LIN {X 0,Y 446.479,Z 402.372,A -85,B 0,C 180,E1 -8668.18,E2 -8668.18} C_VEL
LIN {X 0,Y 446.415,Z 402.374,A -85,B 0,C 180,E1 -8671.301,E2 -8671.301} C_VEL
LIN {X 0,Y 446.426,Z 402.376,A -85,B 0,C 180,E1 -8674.524,E2 -8674.524} C_VEL
LIN {X 0,Y 446.431,Z 402.379,A -85,B 0,C 180,E1 -8678.083,E2 -8678.083} C_VEL
LIN {X 0,Y 446.448,Z 402.406,A -85,B 0,C 180,E1 -8680.922,E2 -8680.922} C_VEL
LIN {X 0,Y 446.858,Z 405.436,A -85,B 0,C 180,E1 -8683.79,E2 -8683.79} C_VEL
LIN {X 0,Y 447.262,Z 408.259,A -85,B 0,C 180,E1 -8686.288,E2 -8686.288} C_VEL
LIN {X 0,Y 447.316,Z 411.248,A -85,B 0,C 180,E1 -8688.71,E2 -8688.71} C_VEL
LIN {X 0,Y 447.118,Z 415.361,A -85,B 0,C 180,E1 -8691.807,E2 -8691.807} C_VEL
LIN {X 0,Y 446.835,Z 419.717,A -85,B 0,C 180,E1 -8694.874,E2 -8694.874} C_VEL
LIN {X 0,Y 446.566,Z 423.896,A -85,B 0,C 180,E1 -8697.651,E2 -8697.651} C_VEL
LIN {X 0,Y 446.285,Z 428.788,A -85,B 0,C 180,E1 -8700.78,E2 -8700.78} C_VEL
LIN {X 0,Y 446.043,Z 433.937,A -85,B 0,C 180,E1 -8703.912,E2 -8703.912} C_VEL
LIN {X 0,Y 445.834,Z 438.832,A -85,B 0,C 180,E1 -8706.791,E2 -8706.791} C_VEL
LIN {X 0,Y 445.676,Z 443.934,A -85,B 0,C 180,E1 -8709.701,E2 -8709.701} C_VEL
LIN {X 0,Y 445.528,Z 449.059,A -85,B 0,C 180,E1 -8712.56,E2 -8712.56} C_VEL
LIN {X 0,Y 445.534,Z 451.508,A -85,B 0,C 180,E1 -8713.873,E2 -8713.873} C_VEL
LIN {X 0,Y 447.627,Z 463.278,A -85,B 0,C 180,E1 -8714.29,E2 -8714.29} C_VEL
LIN {X 0,Y 449.274,Z 475.733,A -85,B 0,C 180,E1 -8714.868,E2 -8714.868} C_VEL
LIN {X 0,Y 448.649,Z 488.448,A -85,B 0,C 180,E1 -8715.601,E2 -8715.601} C_VEL
LIN {X 0,Y 448.166,Z 497.727,A -85,B 0,C 180,E1 -8716.28,E2 -8716.28} C_VEL
LIN {X 0,Y 447.678,Z 506.19,A -85,B 0,C 180,E1 -8717.024,E2 -8717.024} C_VEL
LIN {X 0,Y 447.323,Z 513.287,A -85,B 0,C 180,E1 -8717.755,E2 -8717.755} C_VEL
LIN {X 0,Y 446.729,Z 522.426,A -85,B 0,C 180,E1 -8718.889,E2 -8718.889} C_VEL
LIN {X 0,Y 446.396,Z 528.63,A -85,B 0,C 180,E1 -8719.798,E2 -8719.798} C_VEL
LIN {X 0,Y 446.041,Z 535.168,A -85,B 0,C 180,E1 -8720.935,E2 -8720.935} C_VEL
LIN {X 0,Y 445.849,Z 539.67,A -85,B 0,C 180,E1 -8721.844,E2 -8721.844} C_VEL
LIN {X 0,Y 445.584,Z 545.162,A -85,B 0,C 180,E1 -8723.207,E2 -8723.207} C_VEL
LIN {X 0,Y 445.49,Z 549.484,A -85,B 0,C 180,E1 -8724.569,E2 -8724.569} C_VEL
LIN {X 0,Y 445.419,Z 551.848,A -85,B 0,C 180,E1 -8725.475,E2 -8725.475} C_VEL
LIN {X 0,Y 445.434,Z 555.032,A -85,B 0,C 180,E1 -8727.287,E2 -8727.287} C_VEL
LIN {X 0,Y 445.356,Z 556.087,A -85,B 0,C 180,E1 -8728.191,E2 -8728.191} C_VEL
LIN {X 0,Y 445.339,Z 556.674,A -85,B 0,C 180,E1 -8729.096,E2 -8729.096} C_VEL
LIN {X 0,Y 445.339,Z 556.674,A -85,B 0,C 180,E1 -8730.904,E2 -8730.904} C_VEL
LIN {X 0,Y 445.356,Z 556.087,A -85,B 0,C 180,E1 -8731.809,E2 -8731.809} C_VEL
LIN {X 0,Y 445.434,Z 555.032,A -85,B 0,C 180,E1 -8732.713,E2 -8732.713} C_VEL
LIN {X 0,Y 445.419,Z 551.848,A -85,B 0,C 180,E1 -8734.525,E2 -8734.525} C_VEL
LIN {X 0,Y 445.491,Z 547.64,A -85,B 0,C 180,E1 -8736.069,E2 -8736.069} C_VEL
LIN {X 0,Y 445.668,Z 543.501,A -85,B 0,C 180,E1 -8737.247,E2 -8737.247} C_VEL
LIN {X 0,Y 445.963,Z 537.48,A -85,B 0,C 180,E1 -8738.61,E2 -8738.61} C_VEL
LIN {X 0,Y 446.227,Z 531.382,A -85,B 0,C 180,E1 -8739.748,E2 -8739.748} C_VEL
LIN {X 0,Y 446.532,Z 525.681,A -85,B 0,C 180,E1 -8740.657,E2 -8740.657} C_VEL
LIN {X 0,Y 447.064,Z 517.126,A -85,B 0,C 180,E1 -8741.792,E2 -8741.792} C_VEL
LIN {X 0,Y 447.555,Z 508.945,A -85,B 0,C 180,E1 -8742.7,E2 -8742.7} C_VEL
LIN {X 0,Y 447.937,Z 500.62,A -85,B 0,C 180,E1 -8743.48,E2 -8743.48} C_VEL
LIN {X 0,Y 448.472,Z 491.713,A -85,B 0,C 180,E1 -8744.173,E2 -8744.173} C_VEL
LIN {X 0,Y 448.975,Z 481.953,A -85,B 0,C 180,E1 -8744.794,E2 -8744.794} C_VEL
LIN {X 0,Y 449.187,Z 474.443,A -85,B 0,C 180,E1 -8745.193,E2 -8745.193} C_VEL
LIN {X 0,Y 447.597,Z 463.013,A -85,B 0,C 180,E1 -8745.72,E2 -8745.72} C_VEL
LIN {X 0,Y 445.662,Z 452.543,A -85,B 0,C 180,E1 -8746.094,E2 -8746.094} C_VEL
LIN {X 0,Y 445.535,Z 451.449,A -85,B 0,C 180,E1 -8746.157,E2 -8746.157} C_VEL
LIN {X 0,Y 445.643,Z 445.63,A -85,B 0,C 180,E1 -8749.34,E2 -8749.34} C_VEL
LIN {X 0,Y 445.775,Z 440.518,A -85,B 0,C 180,E1 -8752.233,E2 -8752.233} C_VEL
LIN {X 0,Y 445.947,Z 435.451,A -85,B 0,C 180,E1 -8755.183,E2 -8755.183} C_VEL
LIN {X 0,Y 446.216,Z 430.442,A -85,B 0,C 180,E1 -8758.196,E2 -8758.196} C_VEL
LIN {X 0,Y 446.487,Z 425.503,A -85,B 0,C 180,E1 -8761.294,E2 -8761.294} C_VEL
LIN {X 0,Y 446.768,Z 420.645,A -85,B 0,C 180,E1 -8764.492,E2 -8764.492} C_VEL
LIN {X 0,Y 447.005,Z 417.453,A -85,B 0,C 180,E1 -8766.693,E2 -8766.693} C_VEL
LIN {X 0,Y 447.227,Z 413.373,A -85,B 0,C 180,E1 -8769.644,E2 -8769.644} C_VEL
LIN {X 0,Y 447.365,Z 409.716,A -85,B 0,C 180,E1 -8772.493,E2 -8772.493} C_VEL
LIN {X 0,Y 447.061,Z 406.738,A -85,B 0,C 180,E1 -8775.024,E2 -8775.024} C_VEL
LIN {X 0,Y 446.515,Z 402.871,A -85,B 0,C 180,E1 -8778.618,E2 -8778.618} C_VEL
LIN {X 0,Y 446.448,Z 402.407,A -85,B 0,C 180,E1 -8779.078,E2 -8779.078} C_VEL
LIN {X 0,Y 446.431,Z 402.378,A -85,B 0,C 180,E1 -8781.917,E2 -8781.917} C_VEL
LIN {X 0,Y 446.426,Z 402.378,A -85,B 0,C 180,E1 -8785.476,E2 -8785.476} C_VEL
LIN {X 0,Y 446.415,Z 402.374,A -85,B 0,C 180,E1 -8788.699,E2 -8788.699} C_VEL
LIN {X 0,Y 446.479,Z 402.372,A -85,B 0,C 180,E1 -8791.82,E2 -8791.82} C_VEL
LIN {X 0,Y 446.451,Z 402.369,A -85,B 0,C 180,E1 -8794.847,E2 -8794.847} C_VEL
LIN {X 0,Y 446.441,Z 402.373,A -85,B 0,C 180,E1 -8798.244,E2 -8798.244} C_VEL
LIN {X 0,Y 446.451,Z 402.375,A -85,B 0,C 180,E1 -8801.648,E2 -8801.648} C_VEL
LIN {X 0,Y 446.509,Z 402.362,A -85,B 0,C 180,E1 -8804.479,E2 -8804.479} C_VEL
LIN {X 0,Y 446.51,Z 402.363,A -85,B 0,C 180,E1 -8808.192,E2 -8808.192} C_VEL
LIN {X 0,Y 446.592,Z 402.356,A -85,B 0,C 180,E1 -8811.857,E2 -8811.857} C_VEL
LIN {X 0,Y 446.638,Z 402.345,A -85,B 0,C 180,E1 -8814.582,E2 -8814.582} C_VEL
LIN {X 0,Y 446.701,Z 402.343,A -85,B 0,C 180,E1 -8817.294,E2 -8817.294} C_VEL
LIN {X 0,Y 446.784,Z 402.329,A -85,B 0,C 180,E1 -8819.999,E2 -8819.999} C_VEL
LIN {X 0,Y 446.701,Z 402.338,A -85,B 0,C 180,E1 -8822.705,E2 -8822.705} C_VEL
LIN {X 0,Y 446.639,Z 402.345,A -85,B 0,C 180,E1 -8826.323,E2 -8826.323} C_VEL
LIN {X 0,Y 446.529,Z 402.363,A -85,B 0,C 180,E1 -8829.055,E2 -8829.055} C_VEL
LIN {X 0,Y 446.514,Z 402.363,A -85,B 0,C 180,E1 -8832.729,E2 -8832.729} C_VEL
LIN {X 0,Y 446.487,Z 402.364,A -85,B 0,C 180,E1 -8836.228,E2 -8836.228} C_VEL
LIN {X 0,Y 446.46,Z 402.373,A -85,B 0,C 180,E1 -8839.303,E2 -8839.303} C_VEL
LIN {X 0,Y 446.408,Z 402.374,A -85,B 0,C 180,E1 -8842.2,E2 -8842.2} C_VEL
LIN {X 0,Y 446.449,Z 402.376,A -85,B 0,C 180,E1 -8845.152,E2 -8845.152} C_VEL
LIN {X 0,Y 446.475,Z 402.366,A -85,B 0,C 180,E1 -8848.179,E2 -8848.179} C_VEL
LIN {X 0,Y 446.411,Z 402.377,A -85,B 0,C 180,E1 -8851.3,E2 -8851.3} C_VEL
LIN {X 0,Y 446.422,Z 402.375,A -85,B 0,C 180,E1 -8854.523,E2 -8854.523} C_VEL
LIN {X 0,Y 446.43,Z 402.372,A -85,B 0,C 180,E1 -8858.083,E2 -8858.083} C_VEL
LIN {X 0,Y 446.439,Z 402.376,A -85,B 0,C 180,E1 -8860.921,E2 -8860.921} C_VEL
LIN {X 0,Y 446.437,Z 402.37,A -85,B 0,C 180,E1 -8863.841,E2 -8863.841} C_VEL
LIN {X 0,Y 446.413,Z 402.377,A -85,B 0,C 180,E1 -8866.401,E2 -8866.401} C_VEL
LIN {X 0,Y 446.444,Z 402.37,A -85,B 0,C 180,E1 -8869.803,E2 -8869.803} C_VEL
LIN {X 0,Y 446.421,Z 402.375,A -85,B 0,C 180,E1 -8872.123,E2 -8872.123} C_VEL
LIN {X 0,Y 446.424,Z 402.372,A -85,B 0,C 180,E1 -8875.477,E2 -8875.477} C_VEL
LIN {X 0,Y 446.411,Z 402.379,A -85,B 0,C 180,E1 -8878.7,E2 -8878.7} C_VEL
LIN {X 0,Y 446.479,Z 402.366,A -85,B 0,C 180,E1 -8881.822,E2 -8881.822} C_VEL
LIN {X 0,Y 446.453,Z 402.371,A -85,B 0,C 180,E1 -8884.848,E2 -8884.848} C_VEL
LIN {X 0,Y 446.443,Z 402.376,A -85,B 0,C 180,E1 -8888.245,E2 -8888.245} C_VEL
LIN {X 0,Y 446.453,Z 402.373,A -85,B 0,C 180,E1 -8891.649,E2 -8891.649} C_VEL
LIN {X 0,Y 446.503,Z 402.369,A -85,B 0,C 180,E1 -8894.48,E2 -8894.48} C_VEL
LIN {X 0,Y 446.514,Z 402.368,A -85,B 0,C 180,E1 -8898.193,E2 -8898.193} C_VEL
LIN {X 0,Y 446.596,Z 402.357,A -85,B 0,C 180,E1 -8901.858,E2 -8901.858} C_VEL
LIN {X 0,Y 446.643,Z 402.351,A -85,B 0,C 180,E1 -8904.583,E2 -8904.583} C_VEL
LIN {X 0,Y 446.622,Z 402.351,A -85,B 0,C 180,E1 -8907.011,E2 -8907.011} C_VEL
LIN {X 0,Y 446.104,Z 402.419,A -85,B 0,C 180,E1 -8907.764,E2 -8907.764} C_VEL
LIN {X 0,Y 443.288,Z 402.77,A -85,B 0,C 180,E1 -8908.987,E2 -8908.987} C_VEL
LIN {X 0,Y 440.801,Z 403.08,A -85,B 0,C 180,E1 -8909.974,E2 -8909.974} C_VEL
LIN {X 0,Y 439.712,Z 403.214,A -85,B 0,C 180,E1 -8910.737,E2 -8910.737} C_VEL
LIN {X 0,Y 439.618,Z 403.224,A -85,B 0,C 180,E1 -8910.996,E2 -8910.996} C_VEL
LIN {X 0,Y 439.653,Z 403.22,A -85,B 0,C 180,E1 -8912.749,E2 -8912.749} C_VEL
LIN {X 0,Y 439.615,Z 403.225,A -85,B 0,C 180,E1 -8916.425,E2 -8916.425} C_VEL
LIN {X 0,Y 439.496,Z 403.24,A -85,B 0,C 180,E1 -8919.201,E2 -8919.201} C_VEL
LIN {X 0,Y 439.461,Z 403.243,A -85,B 0,C 180,E1 -8922.937,E2 -8922.937} C_VEL
LIN {X 0,Y 439.443,Z 403.246,A -85,B 0,C 180,E1 -8926.349,E2 -8926.349} C_VEL
LIN {X 0,Y 439.398,Z 403.255,A -85,B 0,C 180,E1 -8929.626,E2 -8929.626} C_VEL
LIN {X 0,Y 439.36,Z 403.252,A -85,B 0,C 180,E1 -8932.575,E2 -8932.575} C_VEL
LIN {X 0,Y 439.401,Z 403.255,A -85,B 0,C 180,E1 -8935.584,E2 -8935.584} C_VEL
LIN {X 0,Y 439.412,Z 403.246,A -85,B 0,C 180,E1 -8938.673,E2 -8938.673} C_VEL
LIN {X 0,Y 439.365,Z 403.253,A -85,B 0,C 180,E1 -8942.03,E2 -8942.03} C_VEL
LIN {X 0,Y 439.39,Z 403.255,A -85,B 0,C 180,E1 -8945.34,E2 -8945.34} C_VEL
LIN {X 0,Y 439.383,Z 403.25,A -85,B 0,C 180,E1 -8948.594,E2 -8948.594} C_VEL
LIN {X 0,Y 439.382,Z 403.256,A -85,B 0,C 180,E1 -8951.257,E2 -8951.257} C_VEL
LIN {X 0,Y 439.398,Z 403.249,A -85,B 0,C 180,E1 -8954.728,E2 -8954.728} C_VEL
LIN {X 0,Y 439.39,Z 403.25,A -85,B 0,C 180,E1 -8957.796,E2 -8957.796} C_VEL
LIN {X 0,Y 439.417,Z 403.245,A -85,B 0,C 180,E1 -8960.227,E2 -8960.227} C_VEL
LIN {X 0,Y 439.368,Z 403.252,A -85,B 0,C 180,E1 -8963.713,E2 -8963.713} C_VEL
LIN {X 0,Y 439.365,Z 403.259,A -85,B 0,C 180,E1 -8967.054,E2 -8967.054} C_VEL
LIN {X 0,Y 439.387,Z 403.249,A -85,B 0,C 180,E1 -8970.275,E2 -8970.275} C_VEL
LIN {X 0,Y 439.424,Z 403.245,A -85,B 0,C 180,E1 -8973.589,E2 -8973.589} C_VEL
LIN {X 0,Y 439.377,Z 403.252,A -85,B 0,C 180,E1 -8976.43,E2 -8976.43} C_VEL
LIN {X 0,Y 439.379,Z 403.251,A -85,B 0,C 180,E1 -8979.397,E2 -8979.397} C_VEL
LIN {X 0,Y 439.422,Z 403.246,A -85,B 0,C 180,E1 -8982.31,E2 -8982.31} C_VEL
LIN {X 0,Y 439.44,Z 403.245,A -85,B 0,C 180,E1 -8985.174,E2 -8985.174} C_VEL
LIN {X 0,Y 439.474,Z 403.238,A -85,B 0,C 180,E1 -8988.002,E2 -8988.002} C_VEL
LIN {X 0,Y 439.539,Z 403.23,A -85,B 0,C 180,E1 -8991.727,E2 -8991.727} C_VEL
LIN {X 0,Y 439.615,Z 403.226,A -85,B 0,C 180,E1 -8994.496,E2 -8994.496} C_VEL
LIN {X 0,Y 439.627,Z 403.222,A -85,B 0,C 180,E1 -8998.168,E2 -8998.168} C_VEL
LIN {X 0,Y 439.755,Z 403.205,A -85,B 0,C 180,E1 -9000.001,E2 -9000.001} C_VEL
LIN {X 0,Y 439.648,Z 403.221,A -85,B 0,C 180,E1 -9002.749,E2 -9002.749} C_VEL
LIN {X 0,Y 439.61,Z 403.229,A -85,B 0,C 180,E1 -9006.426,E2 -9006.426} C_VEL
LIN {X 0,Y 439.492,Z 403.236,A -85,B 0,C 180,E1 -9009.202,E2 -9009.202} C_VEL
LIN {X 0,Y 439.458,Z 403.241,A -85,B 0,C 180,E1 -9012.938,E2 -9012.938} C_VEL
LIN {X 0,Y 439.453,Z 403.247,A -85,B 0,C 180,E1 -9016.355,E2 -9016.355} C_VEL
LIN {X 0,Y 439.395,Z 403.249,A -85,B 0,C 180,E1 -9019.627,E2 -9019.627} C_VEL
LIN {X 0,Y 439.359,Z 403.255,A -85,B 0,C 180,E1 -9022.576,E2 -9022.576} C_VEL
LIN {X 0,Y 439.399,Z 403.249,A -85,B 0,C 180,E1 -9025.586,E2 -9025.586} C_VEL
LIN {X 0,Y 439.419,Z 403.246,A -85,B 0,C 180,E1 -9028.674,E2 -9028.674} C_VEL
LIN {X 0,Y 439.378,Z 403.257,A -85,B 0,C 180,E1 -9032.034,E2 -9032.034} C_VEL
LIN {X 0,Y 439.392,Z 403.249,A -85,B 0,C 180,E1 -9035.342,E2 -9035.342} C_VEL
LIN {X 0,Y 439.392,Z 403.254,A -85,B 0,C 180,E1 -9038.595,E2 -9038.595} C_VEL
LIN {X 0,Y 439.423,Z 403.252,A -85,B 0,C 180,E1 -9039.854,E2 -9039.854} C_VEL
LIN {X 0,Y 439.506,Z 403.944,A -85,B 0,C 180,E1 -9041.276,E2 -9041.276} C_VEL
LIN {X 0,Y 439.999,Z 407.518,A -85,B 0,C 180,E1 -9044.653,E2 -9044.653} C_VEL
LIN {X 0,Y 440.319,Z 410.493,A -85,B 0,C 180,E1 -9047.241,E2 -9047.241} C_VEL
LIN {X 0,Y 440.213,Z 413.996,A -85,B 0,C 180,E1 -9050.025,E2 -9050.025} C_VEL
LIN {X 0,Y 439.986,Z 417.999,A -85,B 0,C 180,E1 -9053.003,E2 -9053.003} C_VEL
LIN {X 0,Y 439.661,Z 422.609,A -85,B 0,C 180,E1 -9056.225,E2 -9056.225} C_VEL
LIN {X 0,Y 439.378,Z 427.108,A -85,B 0,C 180,E1 -9059.214,E2 -9059.214} C_VEL
LIN {X 0,Y 439.097,Z 432.037,A -85,B 0,C 180,E1 -9062.345,E2 -9062.345} C_VEL
LIN {X 0,Y 438.845,Z 437.044,A -85,B 0,C 180,E1 -9065.394,E2 -9065.394} C_VEL
LIN {X 0,Y 438.673,Z 442.114,A -85,B 0,C 180,E1 -9068.378,E2 -9068.378} C_VEL
LIN {X 0,Y 438.543,Z 447.204,A -85,B 0,C 180,E1 -9071.306,E2 -9071.306} C_VEL
LIN {X 0,Y 438.463,Z 451.337,A -85,B 0,C 180,E1 -9073.602,E2 -9073.602} C_VEL
LIN {X 0,Y 440.818,Z 464.467,A -85,B 0,C 180,E1 -9074.088,E2 -9074.088} C_VEL
LIN {X 0,Y 442.36,Z 476.699,A -85,B 0,C 180,E1 -9074.685,E2 -9074.685} C_VEL
LIN {X 0,Y 441.767,Z 488.251,A -85,B 0,C 180,E1 -9075.372,E2 -9075.372} C_VEL
LIN {X 0,Y 441.245,Z 497.529,A -85,B 0,C 180,E1 -9076.06,E2 -9076.06} C_VEL
LIN {X 0,Y 440.68,Z 506.777,A -85,B 0,C 180,E1 -9076.896,E2 -9076.896} C_VEL
LIN {X 0,Y 440.231,Z 515.009,A -85,B 0,C 180,E1 -9077.788,E2 -9077.788} C_VEL
LIN {X 0,Y 439.743,Z 522.229,A -85,B 0,C 180,E1 -9078.71,E2 -9078.71} C_VEL
LIN {X 0,Y 439.374,Z 528.432,A -85,B 0,C 180,E1 -9079.633,E2 -9079.633} C_VEL
LIN {X 0,Y 439.001,Z 534.97,A -85,B 0,C 180,E1 -9080.788,E2 -9080.788} C_VEL
LIN {X 0,Y 438.784,Z 539.472,A -85,B 0,C 180,E1 -9081.712,E2 -9081.712} C_VEL
LIN {X 0,Y 438.516,Z 544.962,A -85,B 0,C 180,E1 -9083.096,E2 -9083.096} C_VEL
LIN {X 0,Y 438.389,Z 549.286,A -85,B 0,C 180,E1 -9084.48,E2 -9084.48} C_VEL
LIN {X 0,Y 438.348,Z 551.651,A -85,B 0,C 180,E1 -9085.402,E2 -9085.402} C_VEL
LIN {X 0,Y 438.342,Z 554.835,A -85,B 0,C 180,E1 -9087.243,E2 -9087.243} C_VEL
LIN {X 0,Y 438.279,Z 555.89,A -85,B 0,C 180,E1 -9088.162,E2 -9088.162} C_VEL
LIN {X 0,Y 438.252,Z 556.477,A -85,B 0,C 180,E1 -9089.081,E2 -9089.081} C_VEL
LIN {X 0,Y 438.252,Z 556.477,A -85,B 0,C 180,E1 -9090.919,E2 -9090.919} C_VEL
LIN {X 0,Y 438.279,Z 555.89,A -85,B 0,C 180,E1 -9091.838,E2 -9091.838} C_VEL
LIN {X 0,Y 438.342,Z 554.835,A -85,B 0,C 180,E1 -9092.757,E2 -9092.757} C_VEL
LIN {X 0,Y 438.348,Z 551.651,A -85,B 0,C 180,E1 -9094.598,E2 -9094.598} C_VEL
LIN {X 0,Y 438.446,Z 546.759,A -85,B 0,C 180,E1 -9096.37,E2 -9096.37} C_VEL
LIN {X 0,Y 438.681,Z 541.388,A -85,B 0,C 180,E1 -9097.826,E2 -9097.826} C_VEL
LIN {X 0,Y 438.97,Z 536.127,A -85,B 0,C 180,E1 -9098.98,E2 -9098.98} C_VEL
LIN {X 0,Y 439.287,Z 529.808,A -85,B 0,C 180,E1 -9100.136,E2 -9100.136} C_VEL
LIN {X 0,Y 439.616,Z 523.855,A -85,B 0,C 180,E1 -9101.06,E2 -9101.06} C_VEL
LIN {X 0,Y 440.097,Z 516.929,A -85,B 0,C 180,E1 -9101.981,E2 -9101.981} C_VEL
LIN {X 0,Y 440.566,Z 509.883,A -85,B 0,C 180,E1 -9102.787,E2 -9102.787} C_VEL
LIN {X 0,Y 440.995,Z 500.869,A -85,B 0,C 180,E1 -9103.657,E2 -9103.657} C_VEL
LIN {X 0,Y 441.558,Z 491.515,A -85,B 0,C 180,E1 -9104.4,E2 -9104.4} C_VEL
LIN {X 0,Y 442.109,Z 481.756,A -85,B 0,C 180,E1 -9105.029,E2 -9105.029} C_VEL
LIN {X 0,Y 442.316,Z 475.532,A -85,B 0,C 180,E1 -9105.375,E2 -9105.375} C_VEL
LIN {X 0,Y 440.609,Z 463.211,A -85,B 0,C 180,E1 -9105.962,E2 -9105.962} C_VEL
LIN {X 0,Y 438.579,Z 452.59,A -85,B 0,C 180,E1 -9106.355,E2 -9106.355} C_VEL
LIN {X 0,Y 438.462,Z 451.337,A -85,B 0,C 180,E1 -9106.399,E2 -9106.399} C_VEL
LIN {X 0,Y 438.565,Z 445.49,A -85,B 0,C 180,E1 -9109.665,E2 -9109.665} C_VEL
LIN {X 0,Y 438.717,Z 440.405,A -85,B 0,C 180,E1 -9112.61,E2 -9112.61} C_VEL
LIN {X 0,Y 438.913,Z 435.364,A -85,B 0,C 180,E1 -9115.615,E2 -9115.615} C_VEL
LIN {X 0,Y 439.166,Z 430.381,A -85,B 0,C 180,E1 -9118.691,E2 -9118.691} C_VEL
LIN {X 0,Y 439.493,Z 425.467,A -85,B 0,C 180,E1 -9121.85,E2 -9121.85} C_VEL
LIN {X 0,Y 439.789,Z 420.639,A -85,B 0,C 180,E1 -9125.119,E2 -9125.119} C_VEL
LIN {X 0,Y 440.007,Z 417.457,A -85,B 0,C 180,E1 -9127.369,E2 -9127.369} C_VEL
LIN {X 0,Y 440.215,Z 413.963,A -85,B 0,C 180,E1 -9129.975,E2 -9129.975} C_VEL
LIN {X 0,Y 440.319,Z 410.485,A -85,B 0,C 180,E1 -9132.759,E2 -9132.759} C_VEL
LIN {X 0,Y 439.995,Z 407.496,A -85,B 0,C 180,E1 -9135.347,E2 -9135.347} C_VEL
LIN {X 0,Y 439.506,Z 403.945,A -85,B 0,C 180,E1 -9138.724,E2 -9138.724} C_VEL
LIN {X 0,Y 439.445,Z 403.248,A -85,B 0,C 180,E1 -9140.229,E2 -9140.229} C_VEL
LIN {X 0,Y 439.373,Z 403.257,A -85,B 0,C 180,E1 -9143.712,E2 -9143.712} C_VEL
LIN {X 0,Y 439.371,Z 403.251,A -85,B 0,C 180,E1 -9147.053,E2 -9147.053} C_VEL
LIN {X 0,Y 439.391,Z 403.252,A -85,B 0,C 180,E1 -9150.274,E2 -9150.274} C_VEL
LIN {X 0,Y 439.428,Z 403.247,A -85,B 0,C 180,E1 -9153.588,E2 -9153.588} C_VEL
LIN {X 0,Y 439.38,Z 403.251,A -85,B 0,C 180,E1 -9156.429,E2 -9156.429} C_VEL
LIN {X 0,Y 439.381,Z 403.252,A -85,B 0,C 180,E1 -9159.396,E2 -9159.396} C_VEL
LIN {X 0,Y 439.425,Z 403.245,A -85,B 0,C 180,E1 -9162.309,E2 -9162.309} C_VEL
LIN {X 0,Y 439.444,Z 403.243,A -85,B 0,C 180,E1 -9165.173,E2 -9165.173} C_VEL
LIN {X 0,Y 439.476,Z 403.241,A -85,B 0,C 180,E1 -9168.001,E2 -9168.001} C_VEL
LIN {X 0,Y 439.54,Z 403.236,A -85,B 0,C 180,E1 -9171.726,E2 -9171.726} C_VEL
LIN {X 0,Y 439.613,Z 403.221,A -85,B 0,C 180,E1 -9174.495,E2 -9174.495} C_VEL
LIN {X 0,Y 439.627,Z 403.22,A -85,B 0,C 180,E1 -9178.167,E2 -9178.167} C_VEL
LIN {X 0,Y 439.755,Z 403.205,A -85,B 0,C 180,E1 -9179.999,E2 -9179.999} C_VEL
LIN {X 0,Y 439.648,Z 403.217,A -85,B 0,C 180,E1 -9182.748,E2 -9182.748} C_VEL
LIN {X 0,Y 439.61,Z 403.221,A -85,B 0,C 180,E1 -9186.425,E2 -9186.425} C_VEL
LIN {X 0,Y 439.491,Z 403.242,A -85,B 0,C 180,E1 -9189.201,E2 -9189.201} C_VEL
LIN {X 0,Y 439.459,Z 403.243,A -85,B 0,C 180,E1 -9192.937,E2 -9192.937} C_VEL
LIN {X 0,Y 439.438,Z 403.242,A -85,B 0,C 180,E1 -9196.349,E2 -9196.349} C_VEL
LIN {X 0,Y 439.393,Z 403.25,A -85,B 0,C 180,E1 -9199.626,E2 -9199.626} C_VEL
LIN {X 0,Y 439.355,Z 403.254,A -85,B 0,C 180,E1 -9202.575,E2 -9202.575} C_VEL
LIN {X 0,Y 439.396,Z 403.249,A -85,B 0,C 180,E1 -9205.585,E2 -9205.585} C_VEL
LIN {X 0,Y 439.416,Z 403.249,A -85,B 0,C 180,E1 -9208.673,E2 -9208.673} C_VEL
LIN {X 0,Y 439.365,Z 403.251,A -85,B 0,C 180,E1 -9211.86,E2 -9211.86} C_VEL
LIN {X 0,Y 439.392,Z 403.252,A -85,B 0,C 180,E1 -9215.156,E2 -9215.156} C_VEL
LIN {X 0,Y 439.391,Z 403.253,A -85,B 0,C 180,E1 -9218.593,E2 -9218.593} C_VEL
LIN {X 0,Y 439.397,Z 403.25,A -85,B 0,C 180,E1 -9221.259,E2 -9221.259} C_VEL
LIN {X 0,Y 439.402,Z 403.255,A -85,B 0,C 180,E1 -9224.728,E2 -9224.728} C_VEL
LIN {X 0,Y 439.39,Z 403.248,A -85,B 0,C 180,E1 -9227.796,E2 -9227.796} C_VEL
LIN {X 0,Y 439.429,Z 403.246,A -85,B 0,C 180,E1 -9230.229,E2 -9230.229} C_VEL
LIN {X 0,Y 439.37,Z 403.251,A -85,B 0,C 180,E1 -9233.713,E2 -9233.713} C_VEL
LIN {X 0,Y 439.366,Z 403.253,A -85,B 0,C 180,E1 -9237.054,E2 -9237.054} C_VEL
LIN {X 0,Y 439.377,Z 403.255,A -85,B 0,C 180,E1 -9240.275,E2 -9240.275} C_VEL
LIN {X 0,Y 439.425,Z 403.244,A -85,B 0,C 180,E1 -9243.397,E2 -9243.397} C_VEL
LIN {X 0,Y 439.383,Z 403.257,A -85,B 0,C 180,E1 -9246.43,E2 -9246.43} C_VEL
LIN {X 0,Y 439.383,Z 403.249,A -85,B 0,C 180,E1 -9249.397,E2 -9249.397} C_VEL
LIN {X 0,Y 439.427,Z 403.251,A -85,B 0,C 180,E1 -9252.31,E2 -9252.31} C_VEL
LIN {X 0,Y 439.443,Z 403.245,A -85,B 0,C 180,E1 -9255.174,E2 -9255.174} C_VEL
LIN {X 0,Y 439.48,Z 403.244,A -85,B 0,C 180,E1 -9258.001,E2 -9258.001} C_VEL
LIN {X 0,Y 439.544,Z 403.235,A -85,B 0,C 180,E1 -9261.726,E2 -9261.726} C_VEL
LIN {X 0,Y 439.618,Z 403.226,A -85,B 0,C 180,E1 -9264.496,E2 -9264.496} C_VEL
LIN {X 0,Y 439.633,Z 403.224,A -85,B 0,C 180,E1 -9268.168,E2 -9268.168} C_VEL
LIN {X 0,Y 439.761,Z 403.21,A -85,B 0,C 180,E1 -9270,E2 -9270} C_VEL
LIN {X 0,Y 439.618,Z 403.224,A -85,B 0,C 180,E1 -9270.996,E2 -9270.996} C_VEL
LIN {X 0,Y 438.903,Z 403.316,A -85,B 0,C 180,E1 -9271.76,E2 -9271.76} C_VEL
LIN {X 0,Y 435.924,Z 403.684,A -85,B 0,C 180,E1 -9272.999,E2 -9272.999} C_VEL
LIN {X 0,Y 433.472,Z 403.992,A -85,B 0,C 180,E1 -9274,E2 -9274} C_VEL
LIN {X 0,Y 432.5,Z 404.112,A -85,B 0,C 180,E1 -9274.774,E2 -9274.774} C_VEL
LIN {X 0,Y 432.463,Z 404.115,A -85,B 0,C 180,E1 -9275.036,E2 -9275.036} C_VEL
LIN {X 0,Y 432.582,Z 404.104,A -85,B 0,C 180,E1 -9277.679,E2 -9277.679} C_VEL
LIN {X 0,Y 432.389,Z 404.126,A -85,B 0,C 180,E1 -9281.247,E2 -9281.247} C_VEL
LIN {X 0,Y 432.369,Z 404.13,A -85,B 0,C 180,E1 -9284.112,E2 -9284.112} C_VEL
LIN {X 0,Y 432.393,Z 404.124,A -85,B 0,C 180,E1 -9287.011,E2 -9287.011} C_VEL
LIN {X 0,Y 432.334,Z 404.131,A -85,B 0,C 180,E1 -9289.96,E2 -9289.96} C_VEL
LIN {X 0,Y 432.314,Z 404.131,A -85,B 0,C 180,E1 -9292.964,E2 -9292.964} C_VEL
LIN {X 0,Y 432.36,Z 404.126,A -85,B 0,C 180,E1 -9296.032,E2 -9296.032} C_VEL
LIN {X 0,Y 432.337,Z 404.13,A -85,B 0,C 180,E1 -9299.187,E2 -9299.187} C_VEL
LIN {X 0,Y 432.317,Z 404.129,A -85,B 0,C 180,E1 -9302.443,E2 -9302.443} C_VEL
LIN {X 0,Y 432.339,Z 404.132,A -85,B 0,C 180,E1 -9305.632,E2 -9305.632} C_VEL
LIN {X 0,Y 432.345,Z 404.127,A -85,B 0,C 180,E1 -9308.716,E2 -9308.716} C_VEL
LIN {X 0,Y 432.327,Z 404.13,A -85,B 0,C 180,E1 -9311.797,E2 -9311.797} C_VEL
LIN {X 0,Y 432.333,Z 404.127,A -85,B 0,C 180,E1 -9314.346,E2 -9314.346} C_VEL
LIN {X 0,Y 432.317,Z 404.134,A -85,B 0,C 180,E1 -9317.015,E2 -9317.015} C_VEL
LIN {X 0,Y 432.325,Z 404.129,A -85,B 0,C 180,E1 -9319.821,E2 -9319.821} C_VEL
LIN {X 0,Y 432.307,Z 404.137,A -85,B 0,C 180,E1 -9323.023,E2 -9323.023} C_VEL
LIN {X 0,Y 432.351,Z 404.125,A -85,B 0,C 180,E1 -9325.996,E2 -9325.996} C_VEL
LIN {X 0,Y 432.386,Z 404.121,A -85,B 0,C 180,E1 -9329.744,E2 -9329.744} C_VEL
LIN {X 0,Y 432.391,Z 404.123,A -85,B 0,C 180,E1 -9333.372,E2 -9333.372} C_VEL
LIN {X 0,Y 432.362,Z 404.124,A -85,B 0,C 180,E1 -9336.023,E2 -9336.023} C_VEL
LIN {X 0,Y 432.341,Z 404.132,A -85,B 0,C 180,E1 -9339.046,E2 -9339.046} C_VEL
LIN {X 0,Y 432.369,Z 404.123,A -85,B 0,C 180,E1 -9342.011,E2 -9342.011} C_VEL
LIN {X 0,Y 432.387,Z 404.126,A -85,B 0,C 180,E1 -9344.927,E2 -9344.927} C_VEL
LIN {X 0,Y 432.45,Z 404.113,A -85,B 0,C 180,E1 -9347.804,E2 -9347.804} C_VEL
LIN {X 0,Y 432.483,Z 404.109,A -85,B 0,C 180,E1 -9351.591,E2 -9351.591} C_VEL
LIN {X 0,Y 432.591,Z 404.1,A -85,B 0,C 180,E1 -9354.407,E2 -9354.407} C_VEL
LIN {X 0,Y 432.597,Z 404.097,A -85,B 0,C 180,E1 -9358.139,E2 -9358.139} C_VEL
LIN {X 0,Y 432.724,Z 404.08,A -85,B 0,C 180,E1 -9360.001,E2 -9360.001} C_VEL
LIN {X 0,Y 432.597,Z 404.098,A -85,B 0,C 180,E1 -9362.794,E2 -9362.794} C_VEL
LIN {X 0,Y 432.564,Z 404.105,A -85,B 0,C 180,E1 -9366.531,E2 -9366.531} C_VEL
LIN {X 0,Y 432.435,Z 404.115,A -85,B 0,C 180,E1 -9369.354,E2 -9369.354} C_VEL
LIN {X 0,Y 432.423,Z 404.118,A -85,B 0,C 180,E1 -9372.804,E2 -9372.804} C_VEL
LIN {X 0,Y 432.416,Z 404.122,A -85,B 0,C 180,E1 -9376.484,E2 -9376.484} C_VEL
LIN {X 0,Y 432.332,Z 404.132,A -85,B 0,C 180,E1 -9379.961,E2 -9379.961} C_VEL
LIN {X 0,Y 432.313,Z 404.13,A -85,B 0,C 180,E1 -9382.965,E2 -9382.965} C_VEL
LIN {X 0,Y 432.359,Z 404.131,A -85,B 0,C 180,E1 -9386.033,E2 -9386.033} C_VEL
LIN {X 0,Y 432.347,Z 404.126,A -85,B 0,C 180,E1 -9389.188,E2 -9389.188} C_VEL
LIN {X 0,Y 432.327,Z 404.132,A -85,B 0,C 180,E1 -9392.295,E2 -9392.295} C_VEL
LIN {X 0,Y 432.337,Z 404.13,A -85,B 0,C 180,E1 -9394.678,E2 -9394.678} C_VEL
LIN {X 0,Y 432.347,Z 404.133,A -85,B 0,C 180,E1 -9398.149,E2 -9398.149} C_VEL
LIN {X 0,Y 432.361,Z 404.131,A -85,B 0,C 180,E1 -9400.185,E2 -9400.185} C_VEL
LIN {X 0,Y 432.74,Z 406.921,A -85,B 0,C 180,E1 -9403.045,E2 -9403.045} C_VEL
LIN {X 0,Y 433.184,Z 409.864,A -85,B 0,C 180,E1 -9405.764,E2 -9405.764} C_VEL
LIN {X 0,Y 433.32,Z 412.863,A -85,B 0,C 180,E1 -9408.321,E2 -9408.321} C_VEL
LIN {X 0,Y 433.082,Z 416.501,A -85,B 0,C 180,E1 -9411.164,E2 -9411.164} C_VEL
LIN {X 0,Y 432.816,Z 420.707,A -85,B 0,C 180,E1 -9414.282,E2 -9414.282} C_VEL
LIN {X 0,Y 432.466,Z 425.599,A -85,B 0,C 180,E1 -9417.678,E2 -9417.678} C_VEL
LIN {X 0,Y 432.161,Z 430.32,A -85,B 0,C 180,E1 -9420.8,E2 -9420.8} C_VEL
LIN {X 0,Y 431.906,Z 435.276,A -85,B 0,C 180,E1 -9423.939,E2 -9423.939} C_VEL
LIN {X 0,Y 431.671,Z 440.291,A -85,B 0,C 180,E1 -9427,E2 -9427} C_VEL
LIN {X 0,Y 431.489,Z 445.351,A -85,B 0,C 180,E1 -9429.999,E2 -9429.999} C_VEL
LIN {X 0,Y 431.374,Z 451.149,A -85,B 0,C 180,E1 -9433.312,E2 -9433.312} C_VEL
LIN {X 0,Y 434.039,Z 465.87,A -85,B 0,C 180,E1 -9433.889,E2 -9433.889} C_VEL
LIN {X 0,Y 435.455,Z 477.53,A -85,B 0,C 180,E1 -9434.496,E2 -9434.496} C_VEL
LIN {X 0,Y 434.89,Z 488.054,A -85,B 0,C 180,E1 -9435.135,E2 -9435.135} C_VEL
LIN {X 0,Y 434.344,Z 497.332,A -85,B 0,C 180,E1 -9435.834,E2 -9435.834} C_VEL
LIN {X 0,Y 433.842,Z 505.423,A -85,B 0,C 180,E1 -9436.564,E2 -9436.564} C_VEL
LIN {X 0,Y 433.413,Z 512.892,A -85,B 0,C 180,E1 -9437.355,E2 -9437.355} C_VEL
LIN {X 0,Y 432.768,Z 522.031,A -85,B 0,C 180,E1 -9438.526,E2 -9438.526} C_VEL
LIN {X 0,Y 432.354,Z 528.234,A -85,B 0,C 180,E1 -9439.463,E2 -9439.463} C_VEL
LIN {X 0,Y 431.958,Z 534.772,A -85,B 0,C 180,E1 -9440.637,E2 -9440.637} C_VEL
LIN {X 0,Y 431.721,Z 539.274,A -85,B 0,C 180,E1 -9441.575,E2 -9441.575} C_VEL
LIN {X 0,Y 431.437,Z 544.765,A -85,B 0,C 180,E1 -9442.983,E2 -9442.983} C_VEL
LIN {X 0,Y 431.292,Z 549.088,A -85,B 0,C 180,E1 -9444.389,E2 -9444.389} C_VEL
LIN {X 0,Y 431.277,Z 551.455,A -85,B 0,C 180,E1 -9445.327,E2 -9445.327} C_VEL
LIN {X 0,Y 431.237,Z 554.638,A -85,B 0,C 180,E1 -9447.198,E2 -9447.198} C_VEL
LIN {X 0,Y 431.203,Z 555.694,A -85,B 0,C 180,E1 -9448.132,E2 -9448.132} C_VEL
LIN {X 0,Y 431.169,Z 556.281,A -85,B 0,C 180,E1 -9449.066,E2 -9449.066} C_VEL
LIN {X 0,Y 431.169,Z 556.281,A -85,B 0,C 180,E1 -9450.934,E2 -9450.934} C_VEL
LIN {X 0,Y 431.203,Z 555.694,A -85,B 0,C 180,E1 -9451.868,E2 -9451.868} C_VEL
LIN {X 0,Y 431.191,Z 553.25,A -85,B 0,C 180,E1 -9453.738,E2 -9453.738} C_VEL
LIN {X 0,Y 431.303,Z 550.305,A -85,B 0,C 180,E1 -9455.142,E2 -9455.142} C_VEL
LIN {X 0,Y 431.378,Z 546.318,A -85,B 0,C 180,E1 -9456.548,E2 -9456.548} C_VEL
LIN {X 0,Y 431.608,Z 541.19,A -85,B 0,C 180,E1 -9457.956,E2 -9457.956} C_VEL
LIN {X 0,Y 431.899,Z 535.928,A -85,B 0,C 180,E1 -9459.129,E2 -9459.129} C_VEL
LIN {X 0,Y 432.253,Z 529.61,A -85,B 0,C 180,E1 -9460.302,E2 -9460.302} C_VEL
LIN {X 0,Y 432.63,Z 523.658,A -85,B 0,C 180,E1 -9461.241,E2 -9461.241} C_VEL
LIN {X 0,Y 433.14,Z 516.731,A -85,B 0,C 180,E1 -9462.177,E2 -9462.177} C_VEL
LIN {X 0,Y 433.636,Z 508.549,A -85,B 0,C 180,E1 -9463.114,E2 -9463.114} C_VEL
LIN {X 0,Y 434.083,Z 500.547,A -85,B 0,C 180,E1 -9463.89,E2 -9463.89} C_VEL
LIN {X 0,Y 434.675,Z 491.317,A -85,B 0,C 180,E1 -9464.633,E2 -9464.633} C_VEL
LIN {X 0,Y 435.229,Z 481.558,A -85,B 0,C 180,E1 -9465.272,E2 -9465.272} C_VEL
LIN {X 0,Y 435.425,Z 476.499,A -85,B 0,C 180,E1 -9465.565,E2 -9465.565} C_VEL
LIN {X 0,Y 433.662,Z 463.306,A -85,B 0,C 180,E1 -9466.215,E2 -9466.215} C_VEL
LIN {X 0,Y 431.478,Z 452.275,A -85,B 0,C 180,E1 -9466.635,E2 -9466.635} C_VEL
LIN {X 0,Y 431.373,Z 451.149,A -85,B 0,C 180,E1 -9466.688,E2 -9466.688} C_VEL
LIN {X 0,Y 431.488,Z 445.35,A -85,B 0,C 180,E1 -9470.001,E2 -9470.001} C_VEL
LIN {X 0,Y 431.671,Z 440.29,A -85,B 0,C 180,E1 -9473,E2 -9473} C_VEL
LIN {X 0,Y 431.905,Z 435.275,A -85,B 0,C 180,E1 -9476.062,E2 -9476.062} C_VEL
LIN {X 0,Y 432.159,Z 430.318,A -85,B 0,C 180,E1 -9479.2,E2 -9479.2} C_VEL
LIN {X 0,Y 432.477,Z 425.432,A -85,B 0,C 180,E1 -9482.429,E2 -9482.429} C_VEL
LIN {X 0,Y 432.82,Z 420.624,A -85,B 0,C 180,E1 -9485.771,E2 -9485.771} C_VEL
LIN {X 0,Y 433.083,Z 416.472,A -85,B 0,C 180,E1 -9488.836,E2 -9488.836} C_VEL
LIN {X 0,Y 433.295,Z 412.781,A -85,B 0,C 180,E1 -9491.744,E2 -9491.744} C_VEL
LIN {X 0,Y 433.105,Z 409.618,A -85,B 0,C 180,E1 -9494.439,E2 -9494.439} C_VEL
LIN {X 0,Y 432.734,Z 406.878,A -85,B 0,C 180,E1 -9496.99,E2 -9496.99} C_VEL
LIN {X 0,Y 432.361,Z 404.131,A -85,B 0,C 180,E1 -9499.815,E2 -9499.815} C_VEL
LIN {X 0,Y 432.312,Z 404.135,A -85,B 0,C 180,E1 -9503.022,E2 -9503.022} C_VEL
LIN {X 0,Y 432.355,Z 404.133,A -85,B 0,C 180,E1 -9505.995,E2 -9505.995} C_VEL
LIN {X 0,Y 432.39,Z 404.125,A -85,B 0,C 180,E1 -9509.743,E2 -9509.743} C_VEL
LIN {X 0,Y 432.394,Z 404.122,A -85,B 0,C 180,E1 -9513.372,E2 -9513.372} C_VEL
LIN {X 0,Y 432.365,Z 404.129,A -85,B 0,C 180,E1 -9516.023,E2 -9516.023} C_VEL
LIN {X 0,Y 432.343,Z 404.127,A -85,B 0,C 180,E1 -9519.045,E2 -9519.045} C_VEL
LIN {X 0,Y 432.372,Z 404.127,A -85,B 0,C 180,E1 -9522.01,E2 -9522.01} C_VEL
LIN {X 0,Y 432.394,Z 404.12,A -85,B 0,C 180,E1 -9524.926,E2 -9524.926} C_VEL
LIN {X 0,Y 432.451,Z 404.119,A -85,B 0,C 180,E1 -9527.803,E2 -9527.803} C_VEL
LIN {X 0,Y 432.484,Z 404.116,A -85,B 0,C 180,E1 -9531.59,E2 -9531.59} C_VEL
LIN {X 0,Y 432.59,Z 404.096,A -85,B 0,C 180,E1 -9534.406,E2 -9534.406} C_VEL
LIN {X 0,Y 432.597,Z 404.095,A -85,B 0,C 180,E1 -9538.137,E2 -9538.137} C_VEL
LIN {X 0,Y 432.724,Z 404.08,A -85,B 0,C 180,E1 -9539.999,E2 -9539.999} C_VEL
LIN {X 0,Y 432.598,Z 404.096,A -85,B 0,C 180,E1 -9542.793,E2 -9542.793} C_VEL
LIN {X 0,Y 432.565,Z 404.099,A -85,B 0,C 180,E1 -9546.53,E2 -9546.53} C_VEL
LIN {X 0,Y 432.434,Z 404.122,A -85,B 0,C 180,E1 -9549.353,E2 -9549.353} C_VEL
LIN {X 0,Y 432.423,Z 404.119,A -85,B 0,C 180,E1 -9552.804,E2 -9552.804} C_VEL
LIN {X 0,Y 432.403,Z 404.119,A -85,B 0,C 180,E1 -9556.479,E2 -9556.479} C_VEL
LIN {X 0,Y 432.329,Z 404.128,A -85,B 0,C 180,E1 -9559.96,E2 -9559.96} C_VEL
LIN {X 0,Y 432.31,Z 404.136,A -85,B 0,C 180,E1 -9562.964,E2 -9562.964} C_VEL
LIN {X 0,Y 432.355,Z 404.125,A -85,B 0,C 180,E1 -9566.032,E2 -9566.032} C_VEL
LIN {X 0,Y 432.343,Z 404.131,A -85,B 0,C 180,E1 -9569.187,E2 -9569.187} C_VEL
LIN {X 0,Y 432.317,Z 404.13,A -85,B 0,C 180,E1 -9572.293,E2 -9572.293} C_VEL
LIN {X 0,Y 432.332,Z 404.132,A -85,B 0,C 180,E1 -9574.677,E2 -9574.677} C_VEL
LIN {X 0,Y 432.345,Z 404.127,A -85,B 0,C 180,E1 -9578.148,E2 -9578.148} C_VEL
LIN {X 0,Y 432.365,Z 404.124,A -85,B 0,C 180,E1 -9581.608,E2 -9581.608} C_VEL
LIN {X 0,Y 432.371,Z 404.126,A -85,B 0,C 180,E1 -9584.342,E2 -9584.342} C_VEL
LIN {X 0,Y 432.327,Z 404.13,A -85,B 0,C 180,E1 -9588.203,E2 -9588.203} C_VEL
LIN {X 0,Y 432.345,Z 404.127,A -85,B 0,C 180,E1 -9591.284,E2 -9591.284} C_VEL
LIN {X 0,Y 432.339,Z 404.132,A -85,B 0,C 180,E1 -9594.368,E2 -9594.368} C_VEL
LIN {X 0,Y 432.317,Z 404.129,A -85,B 0,C 180,E1 -9597.557,E2 -9597.557} C_VEL
LIN {X 0,Y 432.337,Z 404.13,A -85,B 0,C 180,E1 -9600.813,E2 -9600.813} C_VEL
LIN {X 0,Y 432.36,Z 404.126,A -85,B 0,C 180,E1 -9603.968,E2 -9603.968} C_VEL
LIN {X 0,Y 432.315,Z 404.131,A -85,B 0,C 180,E1 -9607.036,E2 -9607.036} C_VEL
LIN {X 0,Y 432.382,Z 404.128,A -85,B 0,C 180,E1 -9610.515,E2 -9610.515} C_VEL
LIN {X 0,Y 432.426,Z 404.123,A -85,B 0,C 180,E1 -9613.961,E2 -9613.961} C_VEL
LIN {X 0,Y 432.455,Z 404.118,A -85,B 0,C 180,E1 -9617.804,E2 -9617.804} C_VEL
LIN {X 0,Y 432.488,Z 404.114,A -85,B 0,C 180,E1 -9621.59,E2 -9621.59} C_VEL
LIN {X 0,Y 432.595,Z 404.1,A -85,B 0,C 180,E1 -9624.406,E2 -9624.406} C_VEL
LIN {X 0,Y 432.602,Z 404.099,A -85,B 0,C 180,E1 -9628.138,E2 -9628.138} C_VEL
LIN {X 0,Y 432.73,Z 404.086,A -85,B 0,C 180,E1 -9630,E2 -9630} C_VEL
LIN {X 0,Y 432.602,Z 404.098,A -85,B 0,C 180,E1 -9632.794,E2 -9632.794} C_VEL
LIN {X 0,Y 432.463,Z 404.115,A -85,B 0,C 180,E1 -9635.036,E2 -9635.036} C_VEL
LIN {X 0,Y 431.904,Z 404.188,A -85,B 0,C 180,E1 -9635.815,E2 -9635.815} C_VEL
LIN {X 0,Y 429.056,Z 404.539,A -85,B 0,C 180,E1 -9637.08,E2 -9637.08} C_VEL
LIN {X 0,Y 426.571,Z 404.851,A -85,B 0,C 180,E1 -9638.101,E2 -9638.101} C_VEL
LIN {X 0,Y 425.49,Z 404.985,A -85,B 0,C 180,E1 -9638.891,E2 -9638.891} C_VEL
LIN {X 0,Y 425.399,Z 404.995,A -85,B 0,C 180,E1 -9639.159,E2 -9639.159} C_VEL
LIN {X 0,Y 425.389,Z 404.996,A -85,B 0,C 180,E1 -9642.904,E2 -9642.904} C_VEL
LIN {X 0,Y 425.357,Z 405,A -85,B 0,C 180,E1 -9646.605,E2 -9646.605} C_VEL
LIN {X 0,Y 425.324,Z 405.008,A -85,B 0,C 180,E1 -9649.635,E2 -9649.635} C_VEL
LIN {X 0,Y 425.302,Z 405.008,A -85,B 0,C 180,E1 -9653.365,E2 -9653.365} C_VEL
LIN {X 0,Y 425.343,Z 404.999,A -85,B 0,C 180,E1 -9656.844,E2 -9656.844} C_VEL
LIN {X 0,Y 425.285,Z 405.01,A -85,B 0,C 180,E1 -9659.719,E2 -9659.719} C_VEL
LIN {X 0,Y 425.276,Z 405.009,A -85,B 0,C 180,E1 -9663.048,E2 -9663.048} C_VEL
LIN {X 0,Y 425.278,Z 405.008,A -85,B 0,C 180,E1 -9665.929,E2 -9665.929} C_VEL
LIN {X 0,Y 425.296,Z 405.008,A -85,B 0,C 180,E1 -9669.044,E2 -9669.044} C_VEL
LIN {X 0,Y 425.271,Z 405.008,A -85,B 0,C 180,E1 -9672.652,E2 -9672.652} C_VEL
LIN {X 0,Y 425.26,Z 405.009,A -85,B 0,C 180,E1 -9676.045,E2 -9676.045} C_VEL
LIN {X 0,Y 425.267,Z 405.009,A -85,B 0,C 180,E1 -9678.621,E2 -9678.621} C_VEL
LIN {X 0,Y 425.301,Z 405.01,A -85,B 0,C 180,E1 -9681.102,E2 -9681.102} C_VEL
LIN {X 0,Y 425.292,Z 405.007,A -85,B 0,C 180,E1 -9684.664,E2 -9684.664} C_VEL
LIN {X 0,Y 425.257,Z 405.009,A -85,B 0,C 180,E1 -9688.073,E2 -9688.073} C_VEL
LIN {X 0,Y 425.329,Z 405.003,A -85,B 0,C 180,E1 -9691.368,E2 -9691.368} C_VEL
LIN {X 0,Y 425.286,Z 405.008,A -85,B 0,C 180,E1 -9694.555,E2 -9694.555} C_VEL
LIN {X 0,Y 425.278,Z 405.007,A -85,B 0,C 180,E1 -9697.661,E2 -9697.661} C_VEL
LIN {X 0,Y 425.353,Z 405.003,A -85,B 0,C 180,E1 -9700.704,E2 -9700.704} C_VEL
LIN {X 0,Y 425.379,Z 404.994,A -85,B 0,C 180,E1 -9703.688,E2 -9703.688} C_VEL
LIN {X 0,Y 425.385,Z 404.996,A -85,B 0,C 180,E1 -9707.096,E2 -9707.096} C_VEL
LIN {X 0,Y 425.392,Z 404.997,A -85,B 0,C 180,E1 -9710.491,E2 -9710.491} C_VEL
LIN {X 0,Y 425.522,Z 404.977,A -85,B 0,C 180,E1 -9713.362,E2 -9713.362} C_VEL
LIN {X 0,Y 425.364,Z 404.996,A -85,B 0,C 180,E1 -9715.262,E2 -9715.262} C_VEL
LIN {X 0,Y 425.567,Z 404.973,A -85,B 0,C 180,E1 -9718.108,E2 -9718.108} C_VEL
LIN {X 0,Y 425.694,Z 404.956,A -85,B 0,C 180,E1 -9720.001,E2 -9720.001} C_VEL
LIN {X 0,Y 425.549,Z 404.976,A -85,B 0,C 180,E1 -9722.84,E2 -9722.84} C_VEL
LIN {X 0,Y 425.522,Z 404.981,A -85,B 0,C 180,E1 -9726.64,E2 -9726.64} C_VEL
LIN {X 0,Y 425.394,Z 404.992,A -85,B 0,C 180,E1 -9729.51,E2 -9729.51} C_VEL
LIN {X 0,Y 425.386,Z 404.994,A -85,B 0,C 180,E1 -9732.904,E2 -9732.904} C_VEL
LIN {X 0,Y 425.363,Z 404.999,A -85,B 0,C 180,E1 -9736.61,E2 -9736.61} C_VEL
LIN {X 0,Y 425.322,Z 405.002,A -85,B 0,C 180,E1 -9739.636,E2 -9739.636} C_VEL
LIN {X 0,Y 425.282,Z 405.011,A -85,B 0,C 180,E1 -9742.34,E2 -9742.34} C_VEL
LIN {X 0,Y 425.289,Z 405.006,A -85,B 0,C 180,E1 -9745.446,E2 -9745.446} C_VEL
LIN {X 0,Y 425.332,Z 405.001,A -85,B 0,C 180,E1 -9748.633,E2 -9748.633} C_VEL
LIN {X 0,Y 425.268,Z 405.014,A -85,B 0,C 180,E1 -9751.927,E2 -9751.927} C_VEL
LIN {X 0,Y 425.296,Z 405.005,A -85,B 0,C 180,E1 -9755.337,E2 -9755.337} C_VEL
LIN {X 0,Y 425.307,Z 405.009,A -85,B 0,C 180,E1 -9759.046,E2 -9759.046} C_VEL
LIN {X 0,Y 425.347,Z 405.172,A -85,B 0,C 180,E1 -9760.121,E2 -9760.121} C_VEL
LIN {X 0,Y 425.776,Z 408.449,A -85,B 0,C 180,E1 -9763.426,E2 -9763.426} C_VEL
LIN {X 0,Y 426.181,Z 411.408,A -85,B 0,C 180,E1 -9766.164,E2 -9766.164} C_VEL
LIN {X 0,Y 426.246,Z 414.431,A -85,B 0,C 180,E1 -9768.737,E2 -9768.737} C_VEL
LIN {X 0,Y 426.042,Z 417.506,A -85,B 0,C 180,E1 -9771.183,E2 -9771.183} C_VEL
LIN {X 0,Y 425.797,Z 421.213,A -85,B 0,C 180,E1 -9773.977,E2 -9773.977} C_VEL
LIN {X 0,Y 425.436,Z 426.023,A -85,B 0,C 180,E1 -9777.405,E2 -9777.405} C_VEL
LIN {X 0,Y 425.141,Z 430.258,A -85,B 0,C 180,E1 -9780.27,E2 -9780.27} C_VEL
LIN {X 0,Y 424.868,Z 435.187,A -85,B 0,C 180,E1 -9783.473,E2 -9783.473} C_VEL
LIN {X 0,Y 424.609,Z 440.175,A -85,B 0,C 180,E1 -9786.595,E2 -9786.595} C_VEL
LIN {X 0,Y 424.436,Z 445.212,A -85,B 0,C 180,E1 -9789.652,E2 -9789.652} C_VEL
LIN {X 0,Y 424.287,Z 450.997,A -85,B 0,C 180,E1 -9793.047,E2 -9793.047} C_VEL
LIN {X 0,Y 426.31,Z 461.847,A -85,B 0,C 180,E1 -9793.454,E2 -9793.454} C_VEL
LIN {X 0,Y 427.769,Z 471.247,A -85,B 0,C 180,E1 -9793.904,E2 -9793.904} C_VEL
LIN {X 0,Y 428.548,Z 478.34,A -85,B 0,C 180,E1 -9794.301,E2 -9794.301} C_VEL
LIN {X 0,Y 428.031,Z 487.857,A -85,B 0,C 180,E1 -9794.891,E2 -9794.891} C_VEL
LIN {X 0,Y 427.449,Z 497.134,A -85,B 0,C 180,E1 -9795.601,E2 -9795.601} C_VEL
LIN {X 0,Y 426.856,Z 506.069,A -85,B 0,C 180,E1 -9796.43,E2 -9796.43} C_VEL
LIN {X 0,Y 426.308,Z 514.614,A -85,B 0,C 180,E1 -9797.383,E2 -9797.383} C_VEL
LIN {X 0,Y 425.795,Z 521.834,A -85,B 0,C 180,E1 -9798.335,E2 -9798.335} C_VEL
LIN {X 0,Y 425.324,Z 528.035,A -85,B 0,C 180,E1 -9799.287,E2 -9799.287} C_VEL
LIN {X 0,Y 424.903,Z 534.573,A -85,B 0,C 180,E1 -9800.48,E2 -9800.48} C_VEL
LIN {X 0,Y 424.685,Z 539.077,A -85,B 0,C 180,E1 -9801.435,E2 -9801.435} C_VEL
LIN {X 0,Y 424.364,Z 544.567,A -85,B 0,C 180,E1 -9802.865,E2 -9802.865} C_VEL
LIN {X 0,Y 424.199,Z 548.89,A -85,B 0,C 180,E1 -9804.295,E2 -9804.295} C_VEL
LIN {X 0,Y 424.207,Z 551.258,A -85,B 0,C 180,E1 -9805.248,E2 -9805.248} C_VEL
LIN {X 0,Y 424.133,Z 554.44,A -85,B 0,C 180,E1 -9807.151,E2 -9807.151} C_VEL
LIN {X 0,Y 424.13,Z 555.497,A -85,B 0,C 180,E1 -9808.101,E2 -9808.101} C_VEL
LIN {X 0,Y 424.089,Z 556.084,A -85,B 0,C 180,E1 -9809.05,E2 -9809.05} C_VEL
LIN {X 0,Y 424.089,Z 556.084,A -85,B 0,C 180,E1 -9810.95,E2 -9810.95} C_VEL
LIN {X 0,Y 424.13,Z 555.497,A -85,B 0,C 180,E1 -9811.899,E2 -9811.899} C_VEL
LIN {X 0,Y 424.102,Z 553.053,A -85,B 0,C 180,E1 -9813.801,E2 -9813.801} C_VEL
LIN {X 0,Y 424.215,Z 550.108,A -85,B 0,C 180,E1 -9815.228,E2 -9815.228} C_VEL
LIN {X 0,Y 424.302,Z 546.12,A -85,B 0,C 180,E1 -9816.658,E2 -9816.658} C_VEL
LIN {X 0,Y 424.552,Z 540.992,A -85,B 0,C 180,E1 -9818.089,E2 -9818.089} C_VEL
LIN {X 0,Y 424.844,Z 535.73,A -85,B 0,C 180,E1 -9819.282,E2 -9819.282} C_VEL
LIN {X 0,Y 425.226,Z 529.412,A -85,B 0,C 180,E1 -9820.475,E2 -9820.475} C_VEL
LIN {X 0,Y 425.655,Z 523.46,A -85,B 0,C 180,E1 -9821.427,E2 -9821.427} C_VEL
LIN {X 0,Y 426.184,Z 516.534,A -85,B 0,C 180,E1 -9822.379,E2 -9822.379} C_VEL
LIN {X 0,Y 426.702,Z 508.351,A -85,B 0,C 180,E1 -9823.331,E2 -9823.331} C_VEL
LIN {X 0,Y 427.222,Z 499.534,A -85,B 0,C 180,E1 -9824.191,E2 -9824.191} C_VEL
LIN {X 0,Y 427.786,Z 491.12,A -85,B 0,C 180,E1 -9824.874,E2 -9824.874} C_VEL
LIN {X 0,Y 428.383,Z 481.361,A -85,B 0,C 180,E1 -9825.522,E2 -9825.522} C_VEL
LIN {X 0,Y 428.394,Z 476.297,A -85,B 0,C 180,E1 -9825.827,E2 -9825.827} C_VEL
LIN {X 0,Y 426.63,Z 463.545,A -85,B 0,C 180,E1 -9826.474,E2 -9826.474} C_VEL
LIN {X 0,Y 424.425,Z 452.195,A -85,B 0,C 180,E1 -9826.917,E2 -9826.917} C_VEL
LIN {X 0,Y 424.285,Z 450.997,A -85,B 0,C 180,E1 -9826.953,E2 -9826.953} C_VEL
LIN {X 0,Y 424.435,Z 445.209,A -85,B 0,C 180,E1 -9830.348,E2 -9830.348} C_VEL
LIN {X 0,Y 424.609,Z 440.173,A -85,B 0,C 180,E1 -9833.405,E2 -9833.405} C_VEL
LIN {X 0,Y 424.896,Z 434.876,A -85,B 0,C 180,E1 -9836.722,E2 -9836.722} C_VEL
LIN {X 0,Y 425.14,Z 430.254,A -85,B 0,C 180,E1 -9839.73,E2 -9839.73} C_VEL
LIN {X 0,Y 425.473,Z 425.394,A -85,B 0,C 180,E1 -9843.03,E2 -9843.03} C_VEL
LIN {X 0,Y 425.837,Z 420.615,A -85,B 0,C 180,E1 -9846.451,E2 -9846.451} C_VEL
LIN {X 0,Y 426.091,Z 417.026,A -85,B 0,C 180,E1 -9849.174,E2 -9849.174} C_VEL
LIN {X 0,Y 426.255,Z 413.396,A -85,B 0,C 180,E1 -9852.102,E2 -9852.102} C_VEL
LIN {X 0,Y 426.04,Z 410.307,A -85,B 0,C 180,E1 -9854.819,E2 -9854.819} C_VEL
LIN {X 0,Y 425.587,Z 406.997,A -85,B 0,C 180,E1 -9857.996,E2 -9857.996} C_VEL
LIN {X 0,Y 425.347,Z 405.177,A -85,B 0,C 180,E1 -9859.879,E2 -9859.879} C_VEL
LIN {X 0,Y 425.282,Z 405.013,A -85,B 0,C 180,E1 -9862.486,E2 -9862.486} C_VEL
LIN {X 0,Y 425.304,Z 405.011,A -85,B 0,C 180,E1 -9865.816,E2 -9865.816} C_VEL
LIN {X 0,Y 425.297,Z 405.004,A -85,B 0,C 180,E1 -9869.235,E2 -9869.235} C_VEL
LIN {X 0,Y 425.345,Z 405,A -85,B 0,C 180,E1 -9872.442,E2 -9872.442} C_VEL
LIN {X 0,Y 425.345,Z 405.002,A -85,B 0,C 180,E1 -9875.601,E2 -9875.601} C_VEL
LIN {X 0,Y 425.286,Z 405.005,A -85,B 0,C 180,E1 -9878.681,E2 -9878.681} C_VEL
LIN {X 0,Y 425.327,Z 405.007,A -85,B 0,C 180,E1 -9881.702,E2 -9881.702} C_VEL
LIN {X 0,Y 425.349,Z 404.997,A -85,B 0,C 180,E1 -9884.67,E2 -9884.67} C_VEL
LIN {X 0,Y 425.404,Z 404.997,A -85,B 0,C 180,E1 -9887.597,E2 -9887.597} C_VEL
LIN {X 0,Y 425.435,Z 404.992,A -85,B 0,C 180,E1 -9891.449,E2 -9891.449} C_VEL
LIN {X 0,Y 425.546,Z 404.973,A -85,B 0,C 180,E1 -9894.313,E2 -9894.313} C_VEL
LIN {X 0,Y 425.567,Z 404.971,A -85,B 0,C 180,E1 -9898.107,E2 -9898.107} C_VEL
LIN {X 0,Y 425.694,Z 404.956,A -85,B 0,C 180,E1 -9899.999,E2 -9899.999} C_VEL
LIN {X 0,Y 425.549,Z 404.974,A -85,B 0,C 180,E1 -9902.839,E2 -9902.839} C_VEL
LIN {X 0,Y 425.522,Z 404.977,A -85,B 0,C 180,E1 -9906.641,E2 -9906.641} C_VEL
LIN {X 0,Y 425.392,Z 404.997,A -85,B 0,C 180,E1 -9909.509,E2 -9909.509} C_VEL
LIN {X 0,Y 425.385,Z 404.996,A -85,B 0,C 180,E1 -9912.904,E2 -9912.904} C_VEL
LIN {X 0,Y 425.352,Z 404.998,A -85,B 0,C 180,E1 -9916.605,E2 -9916.605} C_VEL
LIN {X 0,Y 425.319,Z 405.003,A -85,B 0,C 180,E1 -9919.635,E2 -9919.635} C_VEL
LIN {X 0,Y 425.297,Z 405.008,A -85,B 0,C 180,E1 -9923.365,E2 -9923.365} C_VEL
LIN {X 0,Y 425.34,Z 405.004,A -85,B 0,C 180,E1 -9926.844,E2 -9926.844} C_VEL
LIN {X 0,Y 425.309,Z 405.003,A -85,B 0,C 180,E1 -9929.717,E2 -9929.717} C_VEL
LIN {X 0,Y 425.274,Z 405.013,A -85,B 0,C 180,E1 -9933.048,E2 -9933.048} C_VEL
LIN {X 0,Y 425.276,Z 405.007,A -85,B 0,C 180,E1 -9935.929,E2 -9935.929} C_VEL
LIN {X 0,Y 425.305,Z 405.008,A -85,B 0,C 180,E1 -9939.046,E2 -9939.046} C_VEL
LIN {X 0,Y 425.324,Z 405.007,A -85,B 0,C 180,E1 -9942.646,E2 -9942.646} C_VEL
LIN {X 0,Y 425.261,Z 405.009,A -85,B 0,C 180,E1 -9946.045,E2 -9946.045} C_VEL
LIN {X 0,Y 425.277,Z 405.007,A -85,B 0,C 180,E1 -9949.479,E2 -9949.479} C_VEL
LIN {X 0,Y 425.278,Z 405.012,A -85,B 0,C 180,E1 -9952.488,E2 -9952.488} C_VEL
LIN {X 0,Y 425.301,Z 405.004,A -85,B 0,C 180,E1 -9955.818,E2 -9955.818} C_VEL
LIN {X 0,Y 425.284,Z 405.006,A -85,B 0,C 180,E1 -9959.239,E2 -9959.239} C_VEL
LIN {X 0,Y 425.344,Z 405.006,A -85,B 0,C 180,E1 -9962.443,E2 -9962.443} C_VEL
LIN {X 0,Y 425.346,Z 404.998,A -85,B 0,C 180,E1 -9965.602,E2 -9965.602} C_VEL
LIN {X 0,Y 425.289,Z 405.011,A -85,B 0,C 180,E1 -9968.682,E2 -9968.682} C_VEL
LIN {X 0,Y 425.329,Z 405.005,A -85,B 0,C 180,E1 -9971.703,E2 -9971.703} C_VEL
LIN {X 0,Y 425.344,Z 405.004,A -85,B 0,C 180,E1 -9974.671,E2 -9974.671} C_VEL
LIN {X 0,Y 425.408,Z 404.995,A -85,B 0,C 180,E1 -9977.598,E2 -9977.598} C_VEL
LIN {X 0,Y 425.439,Z 404.992,A -85,B 0,C 180,E1 -9981.45,E2 -9981.45} C_VEL
LIN {X 0,Y 425.551,Z 404.978,A -85,B 0,C 180,E1 -9984.313,E2 -9984.313} C_VEL
LIN {X 0,Y 425.572,Z 404.975,A -85,B 0,C 180,E1 -9988.107,E2 -9988.107} C_VEL
LIN {X 0,Y 425.7,Z 404.961,A -85,B 0,C 180,E1 -9990,E2 -9990} C_VEL
LIN {X 0,Y 425.554,Z 404.976,A -85,B 0,C 180,E1 -9992.84,E2 -9992.84} C_VEL
LIN {X 0,Y 425.528,Z 404.979,A -85,B 0,C 180,E1 -9996.639,E2 -9996.639} C_VEL
LIN {X 0,Y 425.399,Z 404.995,A -85,B 0,C 180,E1 -9999.159,E2 -9999.159} C_VEL
LIN {X 0,Y 424.727,Z 405.082,A -85,B 0,C 180,E1 -9999.949,E2 -9999.949} C_VEL
LIN {X 0,Y 421.879,Z 405.436,A -85,B 0,C 180,E1 -10001.232,E2 -10001.232} C_VEL
LIN {X 0,Y 419.462,Z 405.736,A -85,B 0,C 180,E1 -10002.268,E2 -10002.268} C_VEL
LIN {X 0,Y 418.411,Z 405.866,A -85,B 0,C 180,E1 -10003.069,E2 -10003.069} C_VEL
LIN {X 0,Y 418.318,Z 405.878,A -85,B 0,C 180,E1 -10003.34,E2 -10003.34} C_VEL
LIN {X 0,Y 418.309,Z 405.878,A -85,B 0,C 180,E1 -10006.735,E2 -10006.735} C_VEL
LIN {X 0,Y 418.266,Z 405.886,A -85,B 0,C 180,E1 -10009.79,E2 -10009.79} C_VEL
LIN {X 0,Y 418.233,Z 405.884,A -85,B 0,C 180,E1 -10012.736,E2 -10012.736} C_VEL
LIN {X 0,Y 418.266,Z 405.883,A -85,B 0,C 180,E1 -10015.904,E2 -10015.904} C_VEL
LIN {X 0,Y 418.259,Z 405.884,A -85,B 0,C 180,E1 -10019.162,E2 -10019.162} C_VEL
LIN {X 0,Y 418.251,Z 405.883,A -85,B 0,C 180,E1 -10022.844,E2 -10022.844} C_VEL
LIN {X 0,Y 418.242,Z 405.883,A -85,B 0,C 180,E1 -10026.238,E2 -10026.238} C_VEL
LIN {X 0,Y 418.248,Z 405.885,A -85,B 0,C 180,E1 -10029.681,E2 -10029.681} C_VEL
LIN {X 0,Y 418.225,Z 405.885,A -85,B 0,C 180,E1 -10032.321,E2 -10032.321} C_VEL
LIN {X 0,Y 418.234,Z 405.889,A -85,B 0,C 180,E1 -10035.109,E2 -10035.109} C_VEL
LIN {X 0,Y 418.234,Z 405.885,A -85,B 0,C 180,E1 -10037.767,E2 -10037.767} C_VEL
LIN {X 0,Y 418.249,Z 405.885,A -85,B 0,C 180,E1 -10041.559,E2 -10041.559} C_VEL
LIN {X 0,Y 418.251,Z 405.888,A -85,B 0,C 180,E1 -10045.159,E2 -10045.159} C_VEL
LIN {X 0,Y 418.237,Z 405.886,A -85,B 0,C 180,E1 -10047.472,E2 -10047.472} C_VEL
LIN {X 0,Y 418.268,Z 405.886,A -85,B 0,C 180,E1 -10050.893,E2 -10050.893} C_VEL
LIN {X 0,Y 418.262,Z 405.88,A -85,B 0,C 180,E1 -10054.096,E2 -10054.096} C_VEL
LIN {X 0,Y 418.229,Z 405.888,A -85,B 0,C 180,E1 -10057.264,E2 -10057.264} C_VEL
LIN {X 0,Y 418.274,Z 405.881,A -85,B 0,C 180,E1 -10060.364,E2 -10060.364} C_VEL
LIN {X 0,Y 418.308,Z 405.876,A -85,B 0,C 180,E1 -10063.405,E2 -10063.405} C_VEL
LIN {X 0,Y 418.338,Z 405.875,A -85,B 0,C 180,E1 -10066.999,E2 -10066.999} C_VEL
LIN {X 0,Y 418.332,Z 405.875,A -85,B 0,C 180,E1 -10070.329,E2 -10070.329} C_VEL
LIN {X 0,Y 418.485,Z 405.854,A -85,B 0,C 180,E1 -10073.249,E2 -10073.249} C_VEL
LIN {X 0,Y 418.334,Z 405.873,A -85,B 0,C 180,E1 -10075.182,E2 -10075.182} C_VEL
LIN {X 0,Y 418.536,Z 405.848,A -85,B 0,C 180,E1 -10078.076,E2 -10078.076} C_VEL
LIN {X 0,Y 418.664,Z 405.832,A -85,B 0,C 180,E1 -10080.001,E2 -10080.001} C_VEL
LIN {X 0,Y 418.503,Z 405.853,A -85,B 0,C 180,E1 -10082.888,E2 -10082.888} C_VEL
LIN {X 0,Y 418.485,Z 405.856,A -85,B 0,C 180,E1 -10086.752,E2 -10086.752} C_VEL
LIN {X 0,Y 418.334,Z 405.872,A -85,B 0,C 180,E1 -10089.672,E2 -10089.672} C_VEL
LIN {X 0,Y 418.339,Z 405.872,A -85,B 0,C 180,E1 -10093.001,E2 -10093.001} C_VEL
LIN {X 0,Y 418.313,Z 405.876,A -85,B 0,C 180,E1 -10096.74,E2 -10096.74} C_VEL
LIN {X 0,Y 418.264,Z 405.883,A -85,B 0,C 180,E1 -10099.791,E2 -10099.791} C_VEL
LIN {X 0,Y 418.226,Z 405.886,A -85,B 0,C 180,E1 -10102.737,E2 -10102.737} C_VEL
LIN {X 0,Y 418.265,Z 405.885,A -85,B 0,C 180,E1 -10105.905,E2 -10105.905} C_VEL
LIN {X 0,Y 418.269,Z 405.879,A -85,B 0,C 180,E1 -10109.162,E2 -10109.162} C_VEL
LIN {X 0,Y 418.256,Z 405.881,A -85,B 0,C 180,E1 -10112.845,E2 -10112.845} C_VEL
LIN {X 0,Y 418.245,Z 405.89,A -85,B 0,C 180,E1 -10116.24,E2 -10116.24} C_VEL
LIN {X 0,Y 418.281,Z 405.941,A -85,B 0,C 180,E1 -10119.679,E2 -10119.679} C_VEL
LIN {X 0,Y 418.653,Z 408.528,A -85,B 0,C 180,E1 -10122.386,E2 -10122.386} C_VEL
LIN {X 0,Y 419.075,Z 411.459,A -85,B 0,C 180,E1 -10125.224,E2 -10125.224} C_VEL
LIN {X 0,Y 419.241,Z 414.452,A -85,B 0,C 180,E1 -10127.892,E2 -10127.892} C_VEL
LIN {X 0,Y 419.082,Z 417.591,A -85,B 0,C 180,E1 -10130.482,E2 -10130.482} C_VEL
LIN {X 0,Y 418.743,Z 422.209,A -85,B 0,C 180,E1 -10134.026,E2 -10134.026} C_VEL
LIN {X 0,Y 418.383,Z 426.967,A -85,B 0,C 180,E1 -10137.485,E2 -10137.485} C_VEL
LIN {X 0,Y 418.135,Z 430.196,A -85,B 0,C 180,E1 -10139.72,E2 -10139.72} C_VEL
LIN {X 0,Y 417.856,Z 435.191,A -85,B 0,C 180,E1 -10143.053,E2 -10143.053} C_VEL
LIN {X 0,Y 417.56,Z 440.06,A -85,B 0,C 180,E1 -10146.175,E2 -10146.175} C_VEL
LIN {X 0,Y 417.382,Z 445.07,A -85,B 0,C 180,E1 -10149.293,E2 -10149.293} C_VEL
LIN {X 0,Y 417.197,Z 450.798,A -85,B 0,C 180,E1 -10152.746,E2 -10152.746} C_VEL
LIN {X 0,Y 419.506,Z 462.793,A -85,B 0,C 180,E1 -10153.218,E2 -10153.218} C_VEL
LIN {X 0,Y 421.375,Z 475.787,A -85,B 0,C 180,E1 -10153.885,E2 -10153.885} C_VEL
LIN {X 0,Y 421.587,Z 480.554,A -85,B 0,C 180,E1 -10154.183,E2 -10154.183} C_VEL
LIN {X 0,Y 421.03,Z 489.29,A -85,B 0,C 180,E1 -10154.758,E2 -10154.758} C_VEL
LIN {X 0,Y 420.445,Z 498.288,A -85,B 0,C 180,E1 -10155.479,E2 -10155.479} C_VEL
LIN {X 0,Y 419.865,Z 506.757,A -85,B 0,C 180,E1 -10156.296,E2 -10156.296} C_VEL
LIN {X 0,Y 419.341,Z 514.415,A -85,B 0,C 180,E1 -10157.17,E2 -10157.17} C_VEL
LIN {X 0,Y 418.817,Z 521.636,A -85,B 0,C 180,E1 -10158.138,E2 -10158.138} C_VEL
LIN {X 0,Y 418.321,Z 527.837,A -85,B 0,C 180,E1 -10159.106,E2 -10159.106} C_VEL
LIN {X 0,Y 417.86,Z 534.375,A -85,B 0,C 180,E1 -10160.318,E2 -10160.318} C_VEL
LIN {X 0,Y 417.652,Z 538.879,A -85,B 0,C 180,E1 -10161.289,E2 -10161.289} C_VEL
LIN {X 0,Y 417.291,Z 544.369,A -85,B 0,C 180,E1 -10162.743,E2 -10162.743} C_VEL
LIN {X 0,Y 417.116,Z 548.693,A -85,B 0,C 180,E1 -10164.198,E2 -10164.198} C_VEL
LIN {X 0,Y 417.114,Z 551.06,A -85,B 0,C 180,E1 -10165.167,E2 -10165.167} C_VEL
LIN {X 0,Y 417.03,Z 554.243,A -85,B 0,C 180,E1 -10167.102,E2 -10167.102} C_VEL
LIN {X 0,Y 417.057,Z 555.301,A -85,B 0,C 180,E1 -10168.069,E2 -10168.069} C_VEL
LIN {X 0,Y 417.011,Z 555.888,A -85,B 0,C 180,E1 -10169.034,E2 -10169.034} C_VEL
LIN {X 0,Y 417.011,Z 555.888,A -85,B 0,C 180,E1 -10170.966,E2 -10170.966} C_VEL
LIN {X 0,Y 417.057,Z 555.301,A -85,B 0,C 180,E1 -10171.931,E2 -10171.931} C_VEL
LIN {X 0,Y 417.018,Z 552.856,A -85,B 0,C 180,E1 -10173.865,E2 -10173.865} C_VEL
LIN {X 0,Y 417.13,Z 549.91,A -85,B 0,C 180,E1 -10175.317,E2 -10175.317} C_VEL
LIN {X 0,Y 417.236,Z 545.923,A -85,B 0,C 180,E1 -10176.771,E2 -10176.771} C_VEL
LIN {X 0,Y 417.491,Z 540.794,A -85,B 0,C 180,E1 -10178.226,E2 -10178.226} C_VEL
LIN {X 0,Y 417.801,Z 535.531,A -85,B 0,C 180,E1 -10179.439,E2 -10179.439} C_VEL
LIN {X 0,Y 418.2,Z 529.213,A -85,B 0,C 180,E1 -10180.653,E2 -10180.653} C_VEL
LIN {X 0,Y 418.674,Z 523.263,A -85,B 0,C 180,E1 -10181.621,E2 -10181.621} C_VEL
LIN {X 0,Y 419.216,Z 516.336,A -85,B 0,C 180,E1 -10182.588,E2 -10182.588} C_VEL
LIN {X 0,Y 419.785,Z 508.154,A -85,B 0,C 180,E1 -10183.555,E2 -10183.555} C_VEL
LIN {X 0,Y 420.308,Z 499.47,A -85,B 0,C 180,E1 -10184.417,E2 -10184.417} C_VEL
LIN {X 0,Y 420.925,Z 490.923,A -85,B 0,C 180,E1 -10185.122,E2 -10185.122} C_VEL
LIN {X 0,Y 421.484,Z 482.437,A -85,B 0,C 180,E1 -10185.705,E2 -10185.705} C_VEL
LIN {X 0,Y 421.47,Z 476.783,A -85,B 0,C 180,E1 -10186.053,E2 -10186.053} C_VEL
LIN {X 0,Y 419.679,Z 464.036,A -85,B 0,C 180,E1 -10186.73,E2 -10186.73} C_VEL
LIN {X 0,Y 417.413,Z 452.394,A -85,B 0,C 180,E1 -10187.2,E2 -10187.2} C_VEL
LIN {X 0,Y 417.214,Z 450.769,A -85,B 0,C 180,E1 -10187.271,E2 -10187.271} C_VEL
LIN {X 0,Y 417.381,Z 445.069,A -85,B 0,C 180,E1 -10190.707,E2 -10190.707} C_VEL
LIN {X 0,Y 417.56,Z 440.057,A -85,B 0,C 180,E1 -10193.825,E2 -10193.825} C_VEL
LIN {X 0,Y 417.856,Z 435.094,A -85,B 0,C 180,E1 -10197.008,E2 -10197.008} C_VEL
LIN {X 0,Y 418.136,Z 430.19,A -85,B 0,C 180,E1 -10200.28,E2 -10200.28} C_VEL
LIN {X 0,Y 418.474,Z 425.351,A -85,B 0,C 180,E1 -10203.656,E2 -10203.656} C_VEL
LIN {X 0,Y 418.87,Z 420.607,A -85,B 0,C 180,E1 -10207.158,E2 -10207.158} C_VEL
LIN {X 0,Y 419.087,Z 417.497,A -85,B 0,C 180,E1 -10209.586,E2 -10209.586} C_VEL
LIN {X 0,Y 419.225,Z 414.014,A -85,B 0,C 180,E1 -10212.47,E2 -10212.47} C_VEL
LIN {X 0,Y 418.978,Z 410.99,A -85,B 0,C 180,E1 -10215.209,E2 -10215.209} C_VEL
LIN {X 0,Y 418.6,Z 408.323,A -85,B 0,C 180,E1 -10217.811,E2 -10217.811} C_VEL
LIN {X 0,Y 418.281,Z 405.935,A -85,B 0,C 180,E1 -10220.321,E2 -10220.321} C_VEL
LIN {X 0,Y 418.242,Z 405.89,A -85,B 0,C 180,E1 -10223.975,E2 -10223.975} C_VEL
LIN {X 0,Y 418.256,Z 405.881,A -85,B 0,C 180,E1 -10227.155,E2 -10227.155} C_VEL
LIN {X 0,Y 418.269,Z 405.879,A -85,B 0,C 180,E1 -10230.838,E2 -10230.838} C_VEL
LIN {X 0,Y 418.265,Z 405.885,A -85,B 0,C 180,E1 -10234.095,E2 -10234.095} C_VEL
LIN {X 0,Y 418.226,Z 405.886,A -85,B 0,C 180,E1 -10237.263,E2 -10237.263} C_VEL
LIN {X 0,Y 418.276,Z 405.88,A -85,B 0,C 180,E1 -10240.363,E2 -10240.363} C_VEL
LIN {X 0,Y 418.319,Z 405.877,A -85,B 0,C 180,E1 -10243.404,E2 -10243.404} C_VEL
LIN {X 0,Y 418.339,Z 405.872,A -85,B 0,C 180,E1 -10246.999,E2 -10246.999} C_VEL
LIN {X 0,Y 418.334,Z 405.872,A -85,B 0,C 180,E1 -10250.328,E2 -10250.328} C_VEL
LIN {X 0,Y 418.485,Z 405.856,A -85,B 0,C 180,E1 -10253.248,E2 -10253.248} C_VEL
LIN {X 0,Y 418.334,Z 405.874,A -85,B 0,C 180,E1 -10255.181,E2 -10255.181} C_VEL
LIN {X 0,Y 418.536,Z 405.847,A -85,B 0,C 180,E1 -10258.075,E2 -10258.075} C_VEL
LIN {X 0,Y 418.664,Z 405.832,A -85,B 0,C 180,E1 -10259.999,E2 -10259.999} C_VEL
LIN {X 0,Y 418.503,Z 405.852,A -85,B 0,C 180,E1 -10262.887,E2 -10262.887} C_VEL
LIN {X 0,Y 418.485,Z 405.854,A -85,B 0,C 180,E1 -10266.751,E2 -10266.751} C_VEL
LIN {X 0,Y 418.332,Z 405.875,A -85,B 0,C 180,E1 -10269.671,E2 -10269.671} C_VEL
LIN {X 0,Y 418.338,Z 405.875,A -85,B 0,C 180,E1 -10273.001,E2 -10273.001} C_VEL
LIN {X 0,Y 418.304,Z 405.877,A -85,B 0,C 180,E1 -10276.735,E2 -10276.735} C_VEL
LIN {X 0,Y 418.261,Z 405.881,A -85,B 0,C 180,E1 -10279.79,E2 -10279.79} C_VEL
LIN {X 0,Y 418.229,Z 405.888,A -85,B 0,C 180,E1 -10282.736,E2 -10282.736} C_VEL
LIN {X 0,Y 418.262,Z 405.88,A -85,B 0,C 180,E1 -10285.904,E2 -10285.904} C_VEL
LIN {X 0,Y 418.266,Z 405.885,A -85,B 0,C 180,E1 -10289.161,E2 -10289.161} C_VEL
LIN {X 0,Y 418.249,Z 405.888,A -85,B 0,C 180,E1 -10292.844,E2 -10292.844} C_VEL
LIN {X 0,Y 418.241,Z 405.884,A -85,B 0,C 180,E1 -10296.239,E2 -10296.239} C_VEL
LIN {X 0,Y 418.258,Z 405.881,A -85,B 0,C 180,E1 -10299.68,E2 -10299.68} C_VEL
LIN {X 0,Y 418.277,Z 405.881,A -85,B 0,C 180,E1 -10302.33,E2 -10302.33} C_VEL
LIN {X 0,Y 418.247,Z 405.885,A -85,B 0,C 180,E1 -10305.112,E2 -10305.112} C_VEL
LIN {X 0,Y 418.235,Z 405.884,A -85,B 0,C 180,E1 -10307.767,E2 -10307.767} C_VEL
LIN {X 0,Y 418.253,Z 405.889,A -85,B 0,C 180,E1 -10310.618,E2 -10310.618} C_VEL
LIN {X 0,Y 418.239,Z 405.884,A -85,B 0,C 180,E1 -10313.976,E2 -10313.976} C_VEL
LIN {X 0,Y 418.251,Z 405.883,A -85,B 0,C 180,E1 -10317.156,E2 -10317.156} C_VEL
LIN {X 0,Y 418.263,Z 405.883,A -85,B 0,C 180,E1 -10320.896,E2 -10320.896} C_VEL
LIN {X 0,Y 418.266,Z 405.883,A -85,B 0,C 180,E1 -10324.096,E2 -10324.096} C_VEL
LIN {X 0,Y 418.233,Z 405.884,A -85,B 0,C 180,E1 -10327.264,E2 -10327.264} C_VEL
LIN {X 0,Y 418.279,Z 405.886,A -85,B 0,C 180,E1 -10330.364,E2 -10330.364} C_VEL
LIN {X 0,Y 418.313,Z 405.878,A -85,B 0,C 180,E1 -10333.405,E2 -10333.405} C_VEL
LIN {X 0,Y 418.342,Z 405.874,A -85,B 0,C 180,E1 -10336.999,E2 -10336.999} C_VEL
LIN {X 0,Y 418.338,Z 405.877,A -85,B 0,C 180,E1 -10340.329,E2 -10340.329} C_VEL
LIN {X 0,Y 418.49,Z 405.855,A -85,B 0,C 180,E1 -10343.249,E2 -10343.249} C_VEL
LIN {X 0,Y 418.337,Z 405.876,A -85,B 0,C 180,E1 -10345.182,E2 -10345.182} C_VEL
LIN {X 0,Y 418.541,Z 405.851,A -85,B 0,C 180,E1 -10348.076,E2 -10348.076} C_VEL
LIN {X 0,Y 418.669,Z 405.837,A -85,B 0,C 180,E1 -10350,E2 -10350} C_VEL
LIN {X 0,Y 418.507,Z 405.854,A -85,B 0,C 180,E1 -10352.888,E2 -10352.888} C_VEL
LIN {X 0,Y 418.49,Z 405.855,A -85,B 0,C 180,E1 -10356.751,E2 -10356.751} C_VEL
LIN {X 0,Y 418.338,Z 405.877,A -85,B 0,C 180,E1 -10359.671,E2 -10359.671} C_VEL
LIN {X 0,Y 418.318,Z 405.878,A -85,B 0,C 180,E1 -10363.34,E2 -10363.34} C_VEL
LIN {X 0,Y 417.625,Z 405.968,A -85,B 0,C 180,E1 -10364.144,E2 -10364.144} C_VEL
LIN {X 0,Y 414.746,Z 406.325,A -85,B 0,C 180,E1 -10365.449,E2 -10365.449} C_VEL
LIN {X 0,Y 412.333,Z 406.623,A -85,B 0,C 180,E1 -10366.503,E2 -10366.503} C_VEL
LIN {X 0,Y 411.312,Z 406.751,A -85,B 0,C 180,E1 -10367.318,E2 -10367.318} C_VEL
LIN {X 0,Y 411.235,Z 406.76,A -85,B 0,C 180,E1 -10367.594,E2 -10367.594} C_VEL
LIN {X 0,Y 411.192,Z 406.762,A -85,B 0,C 180,E1 -10371.034,E2 -10371.034} C_VEL
LIN {X 0,Y 411.222,Z 406.758,A -85,B 0,C 180,E1 -10374.215,E2 -10374.215} C_VEL
LIN {X 0,Y 411.253,Z 406.76,A -85,B 0,C 180,E1 -10377.477,E2 -10377.477} C_VEL
LIN {X 0,Y 411.183,Z 406.763,A -85,B 0,C 180,E1 -10380.847,E2 -10380.847} C_VEL
LIN {X 0,Y 411.2,Z 406.76,A -85,B 0,C 180,E1 -10384.333,E2 -10384.333} C_VEL
LIN {X 0,Y 411.194,Z 406.762,A -85,B 0,C 180,E1 -10387.973,E2 -10387.973} C_VEL
LIN {X 0,Y 411.176,Z 406.763,A -85,B 0,C 180,E1 -10390.504,E2 -10390.504} C_VEL
LIN {X 0,Y 411.17,Z 406.769,A -85,B 0,C 180,E1 -10393.133,E2 -10393.133} C_VEL
LIN {X 0,Y 411.165,Z 406.765,A -85,B 0,C 180,E1 -10395.88,E2 -10395.88} C_VEL
LIN {X 0,Y 411.156,Z 406.768,A -85,B 0,C 180,E1 -10398.771,E2 -10398.771} C_VEL
LIN {X 0,Y 411.191,Z 406.761,A -85,B 0,C 180,E1 -10402.027,E2 -10402.027} C_VEL
LIN {X 0,Y 411.197,Z 406.762,A -85,B 0,C 180,E1 -10405.666,E2 -10405.666} C_VEL
LIN {X 0,Y 411.189,Z 406.767,A -85,B 0,C 180,E1 -10409.153,E2 -10409.153} C_VEL
LIN {X 0,Y 411.251,Z 406.756,A -85,B 0,C 180,E1 -10412.522,E2 -10412.522} C_VEL
LIN {X 0,Y 411.218,Z 406.758,A -85,B 0,C 180,E1 -10415.785,E2 -10415.785} C_VEL
LIN {X 0,Y 411.187,Z 406.768,A -85,B 0,C 180,E1 -10418.966,E2 -10418.966} C_VEL
LIN {X 0,Y 411.243,Z 406.755,A -85,B 0,C 180,E1 -10422.085,E2 -10422.085} C_VEL
LIN {X 0,Y 411.254,Z 406.756,A -85,B 0,C 180,E1 -10425.148,E2 -10425.148} C_VEL
LIN {X 0,Y 411.275,Z 406.752,A -85,B 0,C 180,E1 -10428.168,E2 -10428.168} C_VEL
LIN {X 0,Y 411.432,Z 406.733,A -85,B 0,C 180,E1 -10432.189,E2 -10432.189} C_VEL
LIN {X 0,Y 411.468,Z 406.728,A -85,B 0,C 180,E1 -10434.118,E2 -10434.118} C_VEL
LIN {X 0,Y 411.505,Z 406.724,A -85,B 0,C 180,E1 -10438.043,E2 -10438.043} C_VEL
LIN {X 0,Y 411.633,Z 406.708,A -85,B 0,C 180,E1 -10440.001,E2 -10440.001} C_VEL
LIN {X 0,Y 411.459,Z 406.73,A -85,B 0,C 180,E1 -10442.938,E2 -10442.938} C_VEL
LIN {X 0,Y 411.448,Z 406.731,A -85,B 0,C 180,E1 -10446.868,E2 -10446.868} C_VEL
LIN {X 0,Y 411.286,Z 406.751,A -85,B 0,C 180,E1 -10449.839,E2 -10449.839} C_VEL
LIN {X 0,Y 411.298,Z 406.748,A -85,B 0,C 180,E1 -10453.105,E2 -10453.105} C_VEL
LIN {X 0,Y 411.257,Z 406.754,A -85,B 0,C 180,E1 -10456.87,E2 -10456.87} C_VEL
LIN {X 0,Y 411.224,Z 406.762,A -85,B 0,C 180,E1 -10459.988,E2 -10459.988} C_VEL
LIN {X 0,Y 411.191,Z 406.761,A -85,B 0,C 180,E1 -10463.149,E2 -10463.149} C_VEL
LIN {X 0,Y 411.232,Z 406.76,A -85,B 0,C 180,E1 -10466.382,E2 -10466.382} C_VEL
LIN {X 0,Y 411.206,Z 406.763,A -85,B 0,C 180,E1 -10469.713,E2 -10469.713} C_VEL
LIN {X 0,Y 411.203,Z 406.76,A -85,B 0,C 180,E1 -10473.157,E2 -10473.157} C_VEL
LIN {X 0,Y 411.192,Z 406.766,A -85,B 0,C 180,E1 -10476.554,E2 -10476.554} C_VEL
LIN {X 0,Y 411.233,Z 406.763,A -85,B 0,C 180,E1 -10479.223,E2 -10479.223} C_VEL
LIN {X 0,Y 411.695,Z 410.035,A -85,B 0,C 180,E1 -10482.775,E2 -10482.775} C_VEL
LIN {X 0,Y 412.11,Z 413.096,A -85,B 0,C 180,E1 -10485.747,E2 -10485.747} C_VEL
LIN {X 0,Y 412.172,Z 416.341,A -85,B 0,C 180,E1 -10488.613,E2 -10488.613} C_VEL
LIN {X 0,Y 411.928,Z 420.094,A -85,B 0,C 180,E1 -10491.704,E2 -10491.704} C_VEL
LIN {X 0,Y 411.63,Z 423.741,A -85,B 0,C 180,E1 -10494.515,E2 -10494.515} C_VEL
LIN {X 0,Y 411.247,Z 428.521,A -85,B 0,C 180,E1 -10498.011,E2 -10498.011} C_VEL
LIN {X 0,Y 410.951,Z 432.389,A -85,B 0,C 180,E1 -10500.715,E2 -10500.715} C_VEL
LIN {X 0,Y 410.688,Z 436.648,A -85,B 0,C 180,E1 -10503.582,E2 -10503.582} C_VEL
LIN {X 0,Y 410.438,Z 441.616,A -85,B 0,C 180,E1 -10506.807,E2 -10506.807} C_VEL
LIN {X 0,Y 410.254,Z 447.343,A -85,B 0,C 180,E1 -10510.425,E2 -10510.425} C_VEL
LIN {X 0,Y 410.129,Z 450.578,A -85,B 0,C 180,E1 -10512.422,E2 -10512.422} C_VEL
LIN {X 0,Y 412.957,Z 465.582,A -85,B 0,C 180,E1 -10513.056,E2 -10513.056} C_VEL
LIN {X 0,Y 414.545,Z 477.233,A -85,B 0,C 180,E1 -10513.712,E2 -10513.712} C_VEL
LIN {X 0,Y 414.612,Z 482.499,A -85,B 0,C 180,E1 -10514.044,E2 -10514.044} C_VEL
LIN {X 0,Y 413.858,Z 493.968,A -85,B 0,C 180,E1 -10514.865,E2 -10514.865} C_VEL
LIN {X 0,Y 413.044,Z 505.063,A -85,B 0,C 180,E1 -10515.899,E2 -10515.899} C_VEL
LIN {X 0,Y 412.387,Z 514.217,A -85,B 0,C 180,E1 -10516.95,E2 -10516.95} C_VEL
LIN {X 0,Y 411.83,Z 521.438,A -85,B 0,C 180,E1 -10517.934,E2 -10517.934} C_VEL
LIN {X 0,Y 411.329,Z 527.64,A -85,B 0,C 180,E1 -10518.918,E2 -10518.918} C_VEL
LIN {X 0,Y 410.837,Z 534.177,A -85,B 0,C 180,E1 -10520.15,E2 -10520.15} C_VEL
LIN {X 0,Y 410.596,Z 538.681,A -85,B 0,C 180,E1 -10521.139,E2 -10521.139} C_VEL
LIN {X 0,Y 410.213,Z 544.171,A -85,B 0,C 180,E1 -10522.618,E2 -10522.618} C_VEL
LIN {X 0,Y 410.037,Z 548.495,A -85,B 0,C 180,E1 -10524.097,E2 -10524.097} C_VEL
LIN {X 0,Y 410.026,Z 550.863,A -85,B 0,C 180,E1 -10525.084,E2 -10525.084} C_VEL
LIN {X 0,Y 409.936,Z 552.659,A -85,B 0,C 180,E1 -10526.068,E2 -10526.068} C_VEL
LIN {X 0,Y 409.967,Z 555.104,A -85,B 0,C 180,E1 -10528.035,E2 -10528.035} C_VEL
LIN {X 0,Y 409.936,Z 555.691,A -85,B 0,C 180,E1 -10529.018,E2 -10529.018} C_VEL
LIN {X 0,Y 409.936,Z 555.691,A -85,B 0,C 180,E1 -10530.982,E2 -10530.982} C_VEL
LIN {X 0,Y 409.967,Z 555.104,A -85,B 0,C 180,E1 -10531.965,E2 -10531.965} C_VEL
LIN {X 0,Y 409.936,Z 552.659,A -85,B 0,C 180,E1 -10533.932,E2 -10533.932} C_VEL
LIN {X 0,Y 410.026,Z 549.712,A -85,B 0,C 180,E1 -10535.409,E2 -10535.409} C_VEL
LIN {X 0,Y 410.169,Z 545.725,A -85,B 0,C 180,E1 -10536.889,E2 -10536.889} C_VEL
LIN {X 0,Y 410.452,Z 540.596,A -85,B 0,C 180,E1 -10538.368,E2 -10538.368} C_VEL
LIN {X 0,Y 410.768,Z 535.334,A -85,B 0,C 180,E1 -10539.603,E2 -10539.603} C_VEL
LIN {X 0,Y 411.185,Z 529.015,A -85,B 0,C 180,E1 -10540.837,E2 -10540.837} C_VEL
LIN {X 0,Y 411.686,Z 523.065,A -85,B 0,C 180,E1 -10541.821,E2 -10541.821} C_VEL
LIN {X 0,Y 412.256,Z 516.138,A -85,B 0,C 180,E1 -10542.804,E2 -10542.804} C_VEL
LIN {X 0,Y 412.849,Z 507.956,A -85,B 0,C 180,E1 -10543.787,E2 -10543.787} C_VEL
LIN {X 0,Y 413.329,Z 500.698,A -85,B 0,C 180,E1 -10544.533,E2 -10544.533} C_VEL
LIN {X 0,Y 414.067,Z 490.725,A -85,B 0,C 180,E1 -10545.379,E2 -10545.379} C_VEL
LIN {X 0,Y 414.696,Z 480.749,A -85,B 0,C 180,E1 -10546.062,E2 -10546.062} C_VEL
LIN {X 0,Y 414.063,Z 473.211,A -85,B 0,C 180,E1 -10546.527,E2 -10546.527} C_VEL
LIN {X 0,Y 412.344,Z 462.201,A -85,B 0,C 180,E1 -10547.096,E2 -10547.096} C_VEL
LIN {X 0,Y 410.273,Z 451.866,A -85,B 0,C 180,E1 -10547.517,E2 -10547.517} C_VEL
LIN {X 0,Y 410.127,Z 450.578,A -85,B 0,C 180,E1 -10547.578,E2 -10547.578} C_VEL
LIN {X 0,Y 410.242,Z 446.586,A -85,B 0,C 180,E1 -10550.037,E2 -10550.037} C_VEL
LIN {X 0,Y 410.438,Z 441.573,A -85,B 0,C 180,E1 -10553.193,E2 -10553.193} C_VEL
LIN {X 0,Y 410.687,Z 436.633,A -85,B 0,C 180,E1 -10556.418,E2 -10556.418} C_VEL
LIN {X 0,Y 410.992,Z 431.743,A -85,B 0,C 180,E1 -10559.729,E2 -10559.729} C_VEL
LIN {X 0,Y 411.25,Z 428.505,A -85,B 0,C 180,E1 -10561.989,E2 -10561.989} C_VEL
LIN {X 0,Y 411.629,Z 423.716,A -85,B 0,C 180,E1 -10565.485,E2 -10565.485} C_VEL
LIN {X 0,Y 411.931,Z 420.088,A -85,B 0,C 180,E1 -10568.296,E2 -10568.296} C_VEL
LIN {X 0,Y 412.18,Z 415.971,A -85,B 0,C 180,E1 -10571.68,E2 -10571.68} C_VEL
LIN {X 0,Y 412.086,Z 412.972,A -85,B 0,C 180,E1 -10574.365,E2 -10574.365} C_VEL
LIN {X 0,Y 411.694,Z 410.03,A -85,B 0,C 180,E1 -10577.226,E2 -10577.226} C_VEL
LIN {X 0,Y 411.233,Z 406.762,A -85,B 0,C 180,E1 -10580.777,E2 -10580.777} C_VEL
LIN {X 0,Y 411.196,Z 406.769,A -85,B 0,C 180,E1 -10584.47,E2 -10584.47} C_VEL
LIN {X 0,Y 411.167,Z 406.771,A -85,B 0,C 180,E1 -10588.002,E2 -10588.002} C_VEL
LIN {X 0,Y 411.219,Z 406.759,A -85,B 0,C 180,E1 -10591.409,E2 -10591.409} C_VEL
LIN {X 0,Y 411.231,Z 406.756,A -85,B 0,C 180,E1 -10594.706,E2 -10594.706} C_VEL
LIN {X 0,Y 411.198,Z 406.767,A -85,B 0,C 180,E1 -10597.913,E2 -10597.913} C_VEL
LIN {X 0,Y 411.218,Z 406.758,A -85,B 0,C 180,E1 -10601.051,E2 -10601.051} C_VEL
LIN {X 0,Y 411.256,Z 406.756,A -85,B 0,C 180,E1 -10604.131,E2 -10604.131} C_VEL
LIN {X 0,Y 411.296,Z 406.75,A -85,B 0,C 180,E1 -10607.165,E2 -10607.165} C_VEL
LIN {X 0,Y 411.286,Z 406.751,A -85,B 0,C 180,E1 -10610.161,E2 -10610.161} C_VEL
LIN {X 0,Y 411.448,Z 406.731,A -85,B 0,C 180,E1 -10613.132,E2 -10613.132} C_VEL
LIN {X 0,Y 411.305,Z 406.749,A -85,B 0,C 180,E1 -10615.098,E2 -10615.098} C_VEL
LIN {X 0,Y 411.506,Z 406.724,A -85,B 0,C 180,E1 -10618.042,E2 -10618.042} C_VEL
LIN {X 0,Y 411.633,Z 406.708,A -85,B 0,C 180,E1 -10619.999,E2 -10619.999} C_VEL
LIN {X 0,Y 411.459,Z 406.73,A -85,B 0,C 180,E1 -10622.937,E2 -10622.937} C_VEL
LIN {X 0,Y 411.448,Z 406.731,A -85,B 0,C 180,E1 -10626.867,E2 -10626.867} C_VEL
LIN {X 0,Y 411.284,Z 406.751,A -85,B 0,C 180,E1 -10629.838,E2 -10629.838} C_VEL
LIN {X 0,Y 411.297,Z 406.753,A -85,B 0,C 180,E1 -10633.104,E2 -10633.104} C_VEL
LIN {X 0,Y 411.254,Z 406.757,A -85,B 0,C 180,E1 -10636.869,E2 -10636.869} C_VEL
LIN {X 0,Y 411.222,Z 406.758,A -85,B 0,C 180,E1 -10639.987,E2 -10639.987} C_VEL
LIN {X 0,Y 411.194,Z 406.767,A -85,B 0,C 180,E1 -10643.147,E2 -10643.147} C_VEL
LIN {X 0,Y 411.229,Z 406.757,A -85,B 0,C 180,E1 -10646.381,E2 -10646.381} C_VEL
LIN {X 0,Y 411.202,Z 406.76,A -85,B 0,C 180,E1 -10649.712,E2 -10649.712} C_VEL
LIN {X 0,Y 411.198,Z 406.765,A -85,B 0,C 180,E1 -10653.156,E2 -10653.156} C_VEL
LIN {X 0,Y 411.188,Z 406.765,A -85,B 0,C 180,E1 -10656.553,E2 -10656.553} C_VEL
LIN {X 0,Y 411.221,Z 406.758,A -85,B 0,C 180,E1 -10659.731,E2 -10659.731} C_VEL
LIN {X 0,Y 411.214,Z 406.761,A -85,B 0,C 180,E1 -10663.127,E2 -10663.127} C_VEL
LIN {X 0,Y 411.169,Z 406.764,A -85,B 0,C 180,E1 -10665.88,E2 -10665.88} C_VEL
LIN {X 0,Y 411.159,Z 406.771,A -85,B 0,C 180,E1 -10668.772,E2 -10668.772} C_VEL
LIN {X 0,Y 411.204,Z 406.76,A -85,B 0,C 180,E1 -10671.831,E2 -10671.831} C_VEL
LIN {X 0,Y 411.205,Z 406.761,A -85,B 0,C 180,E1 -10675.122,E2 -10675.122} C_VEL
LIN {X 0,Y 411.16,Z 406.767,A -85,B 0,C 180,E1 -10678.003,E2 -10678.003} C_VEL
LIN {X 0,Y 411.212,Z 406.759,A -85,B 0,C 180,E1 -10681.41,E2 -10681.41} C_VEL
LIN {X 0,Y 411.233,Z 406.756,A -85,B 0,C 180,E1 -10683.619,E2 -10683.619} C_VEL
LIN {X 0,Y 411.198,Z 406.762,A -85,B 0,C 180,E1 -10686.853,E2 -10686.853} C_VEL
LIN {X 0,Y 411.21,Z 406.763,A -85,B 0,C 180,E1 -10690.051,E2 -10690.051} C_VEL
LIN {X 0,Y 411.258,Z 406.757,A -85,B 0,C 180,E1 -10693.131,E2 -10693.131} C_VEL
LIN {X 0,Y 411.301,Z 406.752,A -85,B 0,C 180,E1 -10696.896,E2 -10696.896} C_VEL
LIN {X 0,Y 411.289,Z 406.756,A -85,B 0,C 180,E1 -10700.161,E2 -10700.161} C_VEL
LIN {X 0,Y 411.457,Z 406.731,A -85,B 0,C 180,E1 -10703.133,E2 -10703.133} C_VEL
LIN {X 0,Y 411.308,Z 406.752,A -85,B 0,C 180,E1 -10705.099,E2 -10705.099} C_VEL
LIN {X 0,Y 411.511,Z 406.726,A -85,B 0,C 180,E1 -10708.043,E2 -10708.043} C_VEL
LIN {X 0,Y 411.639,Z 406.713,A -85,B 0,C 180,E1 -10710,E2 -10710} C_VEL
LIN {X 0,Y 411.463,Z 406.731,A -85,B 0,C 180,E1 -10712.937,E2 -10712.937} C_VEL
LIN {X 0,Y 411.457,Z 406.731,A -85,B 0,C 180,E1 -10716.867,E2 -10716.867} C_VEL
LIN {X 0,Y 411.289,Z 406.756,A -85,B 0,C 180,E1 -10719.839,E2 -10719.839} C_VEL
LIN {X 0,Y 411.279,Z 406.754,A -85,B 0,C 180,E1 -10723.328,E2 -10723.328} C_VEL
LIN {X 0,Y 411.253,Z 406.758,A -85,B 0,C 180,E1 -10726.889,E2 -10726.889} C_VEL
LIN {X 0,Y 411.235,Z 406.76,A -85,B 0,C 180,E1 -10727.594,E2 -10727.594} C_VEL
LIN {X 0,Y 410.579,Z 406.845,A -85,B 0,C 180,E1 -10728.412,E2 -10728.412} C_VEL
LIN {X 0,Y 407.704,Z 407.204,A -85,B 0,C 180,E1 -10729.74,E2 -10729.74} C_VEL
LIN {X 0,Y 405.264,Z 407.505,A -85,B 0,C 180,E1 -10730.813,E2 -10730.813} C_VEL
LIN {X 0,Y 404.223,Z 407.637,A -85,B 0,C 180,E1 -10731.643,E2 -10731.643} C_VEL
LIN {X 0,Y 404.142,Z 407.639,A -85,B 0,C 180,E1 -10731.924,E2 -10731.924} C_VEL
LIN {X 0,Y 404.211,Z 407.634,A -85,B 0,C 180,E1 -10735.296,E2 -10735.296} C_VEL
LIN {X 0,Y 404.19,Z 407.636,A -85,B 0,C 180,E1 -10737.999,E2 -10737.999} C_VEL
LIN {X 0,Y 404.133,Z 407.647,A -85,B 0,C 180,E1 -10741.558,E2 -10741.558} C_VEL
LIN {X 0,Y 404.179,Z 407.637,A -85,B 0,C 180,E1 -10745.016,E2 -10745.016} C_VEL
LIN {X 0,Y 404.152,Z 407.639,A -85,B 0,C 180,E1 -10748.756,E2 -10748.756} C_VEL
LIN {X 0,Y 404.118,Z 407.646,A -85,B 0,C 180,E1 -10751.6,E2 -10751.6} C_VEL
LIN {X 0,Y 404.143,Z 407.64,A -85,B 0,C 180,E1 -10754.523,E2 -10754.523} C_VEL
LIN {X 0,Y 404.131,Z 407.647,A -85,B 0,C 180,E1 -10757.296,E2 -10757.296} C_VEL
LIN {X 0,Y 404.161,Z 407.637,A -85,B 0,C 180,E1 -10759.955,E2 -10759.955} C_VEL
LIN {X 0,Y 404.131,Z 407.648,A -85,B 0,C 180,E1 -10763.124,E2 -10763.124} C_VEL
LIN {X 0,Y 404.136,Z 407.64,A -85,B 0,C 180,E1 -10766.188,E2 -10766.188} C_VEL
LIN {X 0,Y 404.145,Z 407.64,A -85,B 0,C 180,E1 -10769.716,E2 -10769.716} C_VEL
LIN {X 0,Y 404.187,Z 407.639,A -85,B 0,C 180,E1 -10773.123,E2 -10773.123} C_VEL
LIN {X 0,Y 404.168,Z 407.639,A -85,B 0,C 180,E1 -10775.334,E2 -10775.334} C_VEL
LIN {X 0,Y 404.129,Z 407.644,A -85,B 0,C 180,E1 -10778.581,E2 -10778.581} C_VEL
LIN {X 0,Y 404.201,Z 407.632,A -85,B 0,C 180,E1 -10781.762,E2 -10781.762} C_VEL
LIN {X 0,Y 404.199,Z 407.638,A -85,B 0,C 180,E1 -10784.882,E2 -10784.882} C_VEL
LIN {X 0,Y 404.248,Z 407.627,A -85,B 0,C 180,E1 -10787.959,E2 -10787.959} C_VEL
LIN {X 0,Y 404.396,Z 407.609,A -85,B 0,C 180,E1 -10792.129,E2 -10792.129} C_VEL
LIN {X 0,Y 404.416,Z 407.606,A -85,B 0,C 180,E1 -10794.016,E2 -10794.016} C_VEL
LIN {X 0,Y 404.475,Z 407.599,A -85,B 0,C 180,E1 -10798.009,E2 -10798.009} C_VEL
LIN {X 0,Y 404.603,Z 407.584,A -85,B 0,C 180,E1 -10800.001,E2 -10800.001} C_VEL
LIN {X 0,Y 404.416,Z 407.607,A -85,B 0,C 180,E1 -10802.989,E2 -10802.989} C_VEL
LIN {X 0,Y 404.395,Z 407.609,A -85,B 0,C 180,E1 -10806.988,E2 -10806.988} C_VEL
LIN {X 0,Y 404.251,Z 407.629,A -85,B 0,C 180,E1 -10810.012,E2 -10810.012} C_VEL
LIN {X 0,Y 404.259,Z 407.625,A -85,B 0,C 180,E1 -10813.212,E2 -10813.212} C_VEL
LIN {X 0,Y 404.212,Z 407.631,A -85,B 0,C 180,E1 -10817.009,E2 -10817.009} C_VEL
LIN {X 0,Y 404.157,Z 407.643,A -85,B 0,C 180,E1 -10820.352,E2 -10820.352} C_VEL
LIN {X 0,Y 404.158,Z 407.639,A -85,B 0,C 180,E1 -10823.576,E2 -10823.576} C_VEL
LIN {X 0,Y 404.178,Z 407.638,A -85,B 0,C 180,E1 -10825.767,E2 -10825.767} C_VEL
LIN {X 0,Y 404.193,Z 407.639,A -85,B 0,C 180,E1 -10828,E2 -10828} C_VEL
LIN {X 0,Y 404.141,Z 407.642,A -85,B 0,C 180,E1 -10831.56,E2 -10831.56} C_VEL
LIN {X 0,Y 404.181,Z 407.636,A -85,B 0,C 180,E1 -10835.017,E2 -10835.017} C_VEL
LIN {X 0,Y 404.162,Z 407.643,A -85,B 0,C 180,E1 -10838.757,E2 -10838.757} C_VEL
LIN {X 0,Y 404.532,Z 410.093,A -85,B 0,C 180,E1 -10841.666,E2 -10841.666} C_VEL
LIN {X 0,Y 404.923,Z 413.02,A -85,B 0,C 180,E1 -10844.635,E2 -10844.635} C_VEL
LIN {X 0,Y 405.149,Z 416.011,A -85,B 0,C 180,E1 -10847.429,E2 -10847.429} C_VEL
LIN {X 0,Y 405.025,Z 419.05,A -85,B 0,C 180,E1 -10850.058,E2 -10850.058} C_VEL
LIN {X 0,Y 404.756,Z 422.683,A -85,B 0,C 180,E1 -10853.009,E2 -10853.009} C_VEL
LIN {X 0,Y 404.376,Z 427.297,A -85,B 0,C 180,E1 -10856.537,E2 -10856.537} C_VEL
LIN {X 0,Y 404.011,Z 431.676,A -85,B 0,C 180,E1 -10859.705,E2 -10859.705} C_VEL
LIN {X 0,Y 403.689,Z 436.544,A -85,B 0,C 180,E1 -10863.087,E2 -10863.087} C_VEL
LIN {X 0,Y 403.374,Z 441.5,A -85,B 0,C 180,E1 -10866.377,E2 -10866.377} C_VEL
LIN {X 0,Y 403.17,Z 446.462,A -85,B 0,C 180,E1 -10869.596,E2 -10869.596} C_VEL
LIN {X 0,Y 403.05,Z 450.423,A -85,B 0,C 180,E1 -10872.126,E2 -10872.126} C_VEL
LIN {X 0,Y 405.237,Z 461.582,A -85,B 0,C 180,E1 -10872.579,E2 -10872.579} C_VEL
LIN {X 0,Y 406.902,Z 471.771,A -85,B 0,C 180,E1 -10873.111,E2 -10873.111} C_VEL
LIN {X 0,Y 407.845,Z 480.847,A -85,B 0,C 180,E1 -10873.68,E2 -10873.68} C_VEL
LIN {X 0,Y 407.19,Z 490.527,A -85,B 0,C 180,E1 -10874.355,E2 -10874.355} C_VEL
LIN {X 0,Y 406.461,Z 500.599,A -85,B 0,C 180,E1 -10875.225,E2 -10875.225} C_VEL
LIN {X 0,Y 405.604,Z 512.1,A -85,B 0,C 180,E1 -10876.472,E2 -10876.472} C_VEL
LIN {X 0,Y 404.848,Z 521.24,A -85,B 0,C 180,E1 -10877.722,E2 -10877.722} C_VEL
LIN {X 0,Y 404.331,Z 527.442,A -85,B 0,C 180,E1 -10878.724,E2 -10878.724} C_VEL
LIN {X 0,Y 403.829,Z 533.98,A -85,B 0,C 180,E1 -10879.978,E2 -10879.978} C_VEL
LIN {X 0,Y 403.558,Z 538.484,A -85,B 0,C 180,E1 -10880.983,E2 -10880.983} C_VEL
LIN {X 0,Y 403.16,Z 543.974,A -85,B 0,C 180,E1 -10882.488,E2 -10882.488} C_VEL
LIN {X 0,Y 402.94,Z 548.297,A -85,B 0,C 180,E1 -10883.993,E2 -10883.993} C_VEL
LIN {X 0,Y 402.938,Z 550.665,A -85,B 0,C 180,E1 -10884.997,E2 -10884.997} C_VEL
LIN {X 0,Y 402.857,Z 552.462,A -85,B 0,C 180,E1 -10885.999,E2 -10885.999} C_VEL
LIN {X 0,Y 402.866,Z 554.907,A -85,B 0,C 180,E1 -10888.001,E2 -10888.001} C_VEL
LIN {X 0,Y 402.863,Z 555.495,A -85,B 0,C 180,E1 -10889,E2 -10889} C_VEL
LIN {X 0,Y 402.863,Z 555.495,A -85,B 0,C 180,E1 -10891,E2 -10891} C_VEL
LIN {X 0,Y 402.866,Z 554.907,A -85,B 0,C 180,E1 -10891.999,E2 -10891.999} C_VEL
LIN {X 0,Y 402.857,Z 552.462,A -85,B 0,C 180,E1 -10894.001,E2 -10894.001} C_VEL
LIN {X 0,Y 402.927,Z 549.515,A -85,B 0,C 180,E1 -10895.505,E2 -10895.505} C_VEL
LIN {X 0,Y 403.083,Z 545.527,A -85,B 0,C 180,E1 -10897.01,E2 -10897.01} C_VEL
LIN {X 0,Y 403.395,Z 540.398,A -85,B 0,C 180,E1 -10898.516,E2 -10898.516} C_VEL
LIN {X 0,Y 403.727,Z 535.135,A -85,B 0,C 180,E1 -10899.772,E2 -10899.772} C_VEL
LIN {X 0,Y 404.179,Z 528.817,A -85,B 0,C 180,E1 -10901.027,E2 -10901.027} C_VEL
LIN {X 0,Y 404.707,Z 522.867,A -85,B 0,C 180,E1 -10902.028,E2 -10902.028} C_VEL
LIN {X 0,Y 405.285,Z 515.939,A -85,B 0,C 180,E1 -10903.028,E2 -10903.028} C_VEL
LIN {X 0,Y 405.893,Z 507.757,A -85,B 0,C 180,E1 -10904.028,E2 -10904.028} C_VEL
LIN {X 0,Y 406.506,Z 499.379,A -85,B 0,C 180,E1 -10904.889,E2 -10904.889} C_VEL
LIN {X 0,Y 407.192,Z 490.527,A -85,B 0,C 180,E1 -10905.645,E2 -10905.645} C_VEL
LIN {X 0,Y 407.823,Z 480.848,A -85,B 0,C 180,E1 -10906.321,E2 -10906.321} C_VEL
LIN {X 0,Y 406.901,Z 471.777,A -85,B 0,C 180,E1 -10906.888,E2 -10906.888} C_VEL
LIN {X 0,Y 405.155,Z 461.307,A -85,B 0,C 180,E1 -10907.434,E2 -10907.434} C_VEL
LIN {X 0,Y 403.031,Z 450.39,A -85,B 0,C 180,E1 -10907.895,E2 -10907.895} C_VEL
LIN {X 0,Y 403.169,Z 446.419,A -85,B 0,C 180,E1 -10910.404,E2 -10910.404} C_VEL
LIN {X 0,Y 403.373,Z 441.457,A -85,B 0,C 180,E1 -10913.623,E2 -10913.623} C_VEL
LIN {X 0,Y 403.687,Z 436.54,A -85,B 0,C 180,E1 -10916.913,E2 -10916.913} C_VEL
LIN {X 0,Y 404.011,Z 431.664,A -85,B 0,C 180,E1 -10920.295,E2 -10920.295} C_VEL
LIN {X 0,Y 404.376,Z 427.294,A -85,B 0,C 180,E1 -10923.463,E2 -10923.463} C_VEL
LIN {X 0,Y 404.756,Z 422.675,A -85,B 0,C 180,E1 -10926.991,E2 -10926.991} C_VEL
LIN {X 0,Y 405.055,Z 418.683,A -85,B 0,C 180,E1 -10930.232,E2 -10930.232} C_VEL
LIN {X 0,Y 405.148,Z 415.992,A -85,B 0,C 180,E1 -10932.571,E2 -10932.571} C_VEL
LIN {X 0,Y 404.894,Z 412.999,A -85,B 0,C 180,E1 -10935.369,E2 -10935.369} C_VEL
LIN {X 0,Y 404.491,Z 409.773,A -85,B 0,C 180,E1 -10938.681,E2 -10938.681} C_VEL
LIN {X 0,Y 404.162,Z 407.642,A -85,B 0,C 180,E1 -10941.243,E2 -10941.243} C_VEL
LIN {X 0,Y 404.181,Z 407.64,A -85,B 0,C 180,E1 -10944.983,E2 -10944.983} C_VEL
LIN {X 0,Y 404.144,Z 407.64,A -85,B 0,C 180,E1 -10948.553,E2 -10948.553} C_VEL
LIN {X 0,Y 404.193,Z 407.639,A -85,B 0,C 180,E1 -10952,E2 -10952} C_VEL
LIN {X 0,Y 404.169,Z 407.638,A -85,B 0,C 180,E1 -10955.333,E2 -10955.333} C_VEL
LIN {X 0,Y 404.132,Z 407.641,A -85,B 0,C 180,E1 -10958.58,E2 -10958.58} C_VEL
LIN {X 0,Y 404.204,Z 407.639,A -85,B 0,C 180,E1 -10961.761,E2 -10961.761} C_VEL
LIN {X 0,Y 404.204,Z 407.632,A -85,B 0,C 180,E1 -10964.881,E2 -10964.881} C_VEL
LIN {X 0,Y 404.249,Z 407.63,A -85,B 0,C 180,E1 -10967.958,E2 -10967.958} C_VEL
LIN {X 0,Y 404.398,Z 407.609,A -85,B 0,C 180,E1 -10972.128,E2 -10972.128} C_VEL
LIN {X 0,Y 404.415,Z 407.608,A -85,B 0,C 180,E1 -10974.014,E2 -10974.014} C_VEL
LIN {X 0,Y 404.475,Z 407.6,A -85,B 0,C 180,E1 -10978.008,E2 -10978.008} C_VEL
LIN {X 0,Y 404.603,Z 407.584,A -85,B 0,C 180,E1 -10979.999,E2 -10979.999} C_VEL
LIN {X 0,Y 404.416,Z 407.608,A -85,B 0,C 180,E1 -10982.988,E2 -10982.988} C_VEL
LIN {X 0,Y 404.388,Z 407.609,A -85,B 0,C 180,E1 -10986.646,E2 -10986.646} C_VEL
LIN {X 0,Y 404.283,Z 407.625,A -85,B 0,C 180,E1 -10989.001,E2 -10989.001} C_VEL
LIN {X 0,Y 404.248,Z 407.627,A -85,B 0,C 180,E1 -10992.041,E2 -10992.041} C_VEL
LIN {X 0,Y 404.199,Z 407.638,A -85,B 0,C 180,E1 -10995.118,E2 -10995.118} C_VEL
LIN {X 0,Y 404.201,Z 407.632,A -85,B 0,C 180,E1 -10998.238,E2 -10998.238} C_VEL
LIN {X 0,Y 404.129,Z 407.644,A -85,B 0,C 180,E1 -11001.419,E2 -11001.419} C_VEL
LIN {X 0,Y 404.168,Z 407.639,A -85,B 0,C 180,E1 -11004.666,E2 -11004.666} C_VEL
LIN {X 0,Y 404.189,Z 407.633,A -85,B 0,C 180,E1 -11007.999,E2 -11007.999} C_VEL
LIN {X 0,Y 404.134,Z 407.641,A -85,B 0,C 180,E1 -11011.559,E2 -11011.559} C_VEL
LIN {X 0,Y 404.177,Z 407.641,A -85,B 0,C 180,E1 -11015.016,E2 -11015.016} C_VEL
LIN {X 0,Y 404.156,Z 407.644,A -85,B 0,C 180,E1 -11018.756,E2 -11018.756} C_VEL
LIN {X 0,Y 404.184,Z 407.634,A -85,B 0,C 180,E1 -11021.611,E2 -11021.611} C_VEL
LIN {X 0,Y 404.183,Z 407.639,A -85,B 0,C 180,E1 -11024.529,E2 -11024.529} C_VEL
LIN {X 0,Y 404.132,Z 407.642,A -85,B 0,C 180,E1 -11027.296,E2 -11027.296} C_VEL
LIN {X 0,Y 404.162,Z 407.638,A -85,B 0,C 180,E1 -11029.956,E2 -11029.956} C_VEL
LIN {X 0,Y 404.133,Z 407.642,A -85,B 0,C 180,E1 -11033.125,E2 -11033.125} C_VEL
LIN {X 0,Y 404.139,Z 407.643,A -85,B 0,C 180,E1 -11036.188,E2 -11036.188} C_VEL
LIN {X 0,Y 404.14,Z 407.64,A -85,B 0,C 180,E1 -11039.715,E2 -11039.715} C_VEL
LIN {X 0,Y 404.19,Z 407.634,A -85,B 0,C 180,E1 -11043.123,E2 -11043.123} C_VEL
LIN {X 0,Y 404.172,Z 407.636,A -85,B 0,C 180,E1 -11045.335,E2 -11045.335} C_VEL
LIN {X 0,Y 404.134,Z 407.646,A -85,B 0,C 180,E1 -11048.581,E2 -11048.581} C_VEL
LIN {X 0,Y 404.206,Z 407.637,A -85,B 0,C 180,E1 -11051.762,E2 -11051.762} C_VEL
LIN {X 0,Y 404.202,Z 407.636,A -85,B 0,C 180,E1 -11054.882,E2 -11054.882} C_VEL
LIN {X 0,Y 404.253,Z 407.632,A -85,B 0,C 180,E1 -11057.959,E2 -11057.959} C_VEL
LIN {X 0,Y 404.429,Z 407.609,A -85,B 0,C 180,E1 -11062.1,E2 -11062.1} C_VEL
LIN {X 0,Y 404.421,Z 407.61,A -85,B 0,C 180,E1 -11064.015,E2 -11064.015} C_VEL
LIN {X 0,Y 404.479,Z 407.602,A -85,B 0,C 180,E1 -11068.009,E2 -11068.009} C_VEL
LIN {X 0,Y 404.608,Z 407.589,A -85,B 0,C 180,E1 -11070,E2 -11070} C_VEL
LIN {X 0,Y 404.42,Z 407.609,A -85,B 0,C 180,E1 -11072.988,E2 -11072.988} C_VEL
LIN {X 0,Y 404.408,Z 407.61,A -85,B 0,C 180,E1 -11076.987,E2 -11076.987} C_VEL
LIN {X 0,Y 404.255,Z 407.632,A -85,B 0,C 180,E1 -11080.012,E2 -11080.012} C_VEL
LIN {X 0,Y 404.262,Z 407.629,A -85,B 0,C 180,E1 -11083.211,E2 -11083.211} C_VEL
LIN {X 0,Y 404.211,Z 407.635,A -85,B 0,C 180,E1 -11087.007,E2 -11087.007} C_VEL
LIN {X 0,Y 404.159,Z 407.638,A -85,B 0,C 180,E1 -11090.351,E2 -11090.351} C_VEL
LIN {X 0,Y 404.142,Z 407.639,A -85,B 0,C 180,E1 -11091.924,E2 -11091.924} C_VEL
LIN {X 0,Y 403.489,Z 407.721,A -85,B 0,C 180,E1 -11092.756,E2 -11092.756} C_VEL
LIN {X 0,Y 400.651,Z 408.076,A -85,B 0,C 180,E1 -11094.107,E2 -11094.107} C_VEL
LIN {X 0,Y 398.244,Z 408.377,A -85,B 0,C 180,E1 -11095.199,E2 -11095.199} C_VEL
LIN {X 0,Y 397.212,Z 408.505,A -85,B 0,C 180,E1 -11096.043,E2 -11096.043} C_VEL
LIN {X 0,Y 397.129,Z 408.513,A -85,B 0,C 180,E1 -11096.329,E2 -11096.329} C_VEL
LIN {X 0,Y 397.116,Z 408.515,A -85,B 0,C 180,E1 -11098.543,E2 -11098.543} C_VEL
LIN {X 0,Y 397.072,Z 408.521,A -85,B 0,C 180,E1 -11102.071,E2 -11102.071} C_VEL
LIN {X 0,Y 397.114,Z 408.521,A -85,B 0,C 180,E1 -11105.503,E2 -11105.503} C_VEL
LIN {X 0,Y 397.127,Z 408.515,A -85,B 0,C 180,E1 -11108.862,E2 -11108.862} C_VEL
LIN {X 0,Y 397.064,Z 408.521,A -85,B 0,C 180,E1 -11112.267,E2 -11112.267} C_VEL
LIN {X 0,Y 397.084,Z 408.523,A -85,B 0,C 180,E1 -11115.068,E2 -11115.068} C_VEL
LIN {X 0,Y 397.06,Z 408.522,A -85,B 0,C 180,E1 -11118.021,E2 -11118.021} C_VEL
LIN {X 0,Y 397.123,Z 408.521,A -85,B 0,C 180,E1 -11121.138,E2 -11121.138} C_VEL
LIN {X 0,Y 397.112,Z 408.516,A -85,B 0,C 180,E1 -11124.496,E2 -11124.496} C_VEL
LIN {X 0,Y 397.072,Z 408.52,A -85,B 0,C 180,E1 -11127.929,E2 -11127.929} C_VEL
LIN {X 0,Y 397.118,Z 408.516,A -85,B 0,C 180,E1 -11131.457,E2 -11131.457} C_VEL
LIN {X 0,Y 397.144,Z 408.513,A -85,B 0,C 180,E1 -11134.488,E2 -11134.488} C_VEL
LIN {X 0,Y 397.1,Z 408.521,A -85,B 0,C 180,E1 -11137.086,E2 -11137.086} C_VEL
LIN {X 0,Y 397.139,Z 408.513,A -85,B 0,C 180,E1 -11140.353,E2 -11140.353} C_VEL
LIN {X 0,Y 397.158,Z 408.51,A -85,B 0,C 180,E1 -11143.553,E2 -11143.553} C_VEL
LIN {X 0,Y 397.22,Z 408.508,A -85,B 0,C 180,E1 -11146.703,E2 -11146.703} C_VEL
LIN {X 0,Y 397.209,Z 408.503,A -85,B 0,C 180,E1 -11149.809,E2 -11149.809} C_VEL
LIN {X 0,Y 397.345,Z 408.49,A -85,B 0,C 180,E1 -11152.888,E2 -11152.888} C_VEL
LIN {X 0,Y 397.249,Z 408.502,A -85,B 0,C 180,E1 -11154.926,E2 -11154.926} C_VEL
LIN {X 0,Y 397.443,Z 408.475,A -85,B 0,C 180,E1 -11157.974,E2 -11157.974} C_VEL
LIN {X 0,Y 397.572,Z 408.459,A -85,B 0,C 180,E1 -11160.001,E2 -11160.001} C_VEL
LIN {X 0,Y 397.374,Z 408.484,A -85,B 0,C 180,E1 -11163.042,E2 -11163.042} C_VEL
LIN {X 0,Y 397.366,Z 408.487,A -85,B 0,C 180,E1 -11166.092,E2 -11166.092} C_VEL
LIN {X 0,Y 397.245,Z 408.499,A -85,B 0,C 180,E1 -11169.163,E2 -11169.163} C_VEL
LIN {X 0,Y 397.212,Z 408.509,A -85,B 0,C 180,E1 -11172.259,E2 -11172.259} C_VEL
LIN {X 0,Y 397.177,Z 408.507,A -85,B 0,C 180,E1 -11175.393,E2 -11175.393} C_VEL
LIN {X 0,Y 397.156,Z 408.513,A -85,B 0,C 180,E1 -11178.574,E2 -11178.574} C_VEL
LIN {X 0,Y 397.089,Z 408.521,A -85,B 0,C 180,E1 -11181.819,E2 -11181.819} C_VEL
LIN {X 0,Y 397.147,Z 408.512,A -85,B 0,C 180,E1 -11185.513,E2 -11185.513} C_VEL
LIN {X 0,Y 397.121,Z 408.516,A -85,B 0,C 180,E1 -11188.544,E2 -11188.544} C_VEL
LIN {X 0,Y 397.107,Z 408.522,A -85,B 0,C 180,E1 -11192.07,E2 -11192.07} C_VEL
LIN {X 0,Y 397.116,Z 408.517,A -85,B 0,C 180,E1 -11195.504,E2 -11195.504} C_VEL
LIN {X 0,Y 397.141,Z 408.729,A -85,B 0,C 180,E1 -11198.865,E2 -11198.865} C_VEL
LIN {X 0,Y 397.598,Z 411.725,A -85,B 0,C 180,E1 -11202.199,E2 -11202.199} C_VEL
LIN {X 0,Y 397.955,Z 414.519,A -85,B 0,C 180,E1 -11205.058,E2 -11205.058} C_VEL
LIN {X 0,Y 398.124,Z 417.518,A -85,B 0,C 180,E1 -11207.872,E2 -11207.872} C_VEL
LIN {X 0,Y 397.912,Z 421.153,A -85,B 0,C 180,E1 -11211,E2 -11211} C_VEL
LIN {X 0,Y 397.551,Z 425.234,A -85,B 0,C 180,E1 -11214.312,E2 -11214.312} C_VEL
LIN {X 0,Y 397.281,Z 428.4,A -85,B 0,C 180,E1 -11216.744,E2 -11216.744} C_VEL
LIN {X 0,Y 397.02,Z 431.595,A -85,B 0,C 180,E1 -11219.113,E2 -11219.113} C_VEL
LIN {X 0,Y 396.671,Z 436.449,A -85,B 0,C 180,E1 -11222.571,E2 -11222.571} C_VEL
LIN {X 0,Y 396.335,Z 441.356,A -85,B 0,C 180,E1 -11225.931,E2 -11225.931} C_VEL
LIN {X 0,Y 396.102,Z 446.322,A -85,B 0,C 180,E1 -11229.216,E2 -11229.216} C_VEL
LIN {X 0,Y 395.95,Z 450.235,A -85,B 0,C 180,E1 -11231.797,E2 -11231.797} C_VEL
LIN {X 0,Y 398.05,Z 460.658,A -85,B 0,C 180,E1 -11232.227,E2 -11232.227} C_VEL
LIN {X 0,Y 399.78,Z 470.661,A -85,B 0,C 180,E1 -11232.755,E2 -11232.755} C_VEL
LIN {X 0,Y 400.951,Z 480.937,A -85,B 0,C 180,E1 -11233.41,E2 -11233.41} C_VEL
LIN {X 0,Y 400.356,Z 490.33,A -85,B 0,C 180,E1 -11234.081,E2 -11234.081} C_VEL
LIN {X 0,Y 399.578,Z 500.402,A -85,B 0,C 180,E1 -11234.964,E2 -11234.964} C_VEL
LIN {X 0,Y 398.624,Z 512.027,A -85,B 0,C 180,E1 -11236.248,E2 -11236.248} C_VEL
LIN {X 0,Y 397.889,Z 521.042,A -85,B 0,C 180,E1 -11237.504,E2 -11237.504} C_VEL
LIN {X 0,Y 397.313,Z 527.243,A -85,B 0,C 180,E1 -11238.522,E2 -11238.522} C_VEL
LIN {X 0,Y 396.811,Z 533.782,A -85,B 0,C 180,E1 -11239.799,E2 -11239.799} C_VEL
LIN {X 0,Y 396.514,Z 538.286,A -85,B 0,C 180,E1 -11240.821,E2 -11240.821} C_VEL
LIN {X 0,Y 396.091,Z 543.776,A -85,B 0,C 180,E1 -11242.353,E2 -11242.353} C_VEL
LIN {X 0,Y 395.863,Z 548.1,A -85,B 0,C 180,E1 -11243.885,E2 -11243.885} C_VEL
LIN {X 0,Y 395.851,Z 550.468,A -85,B 0,C 180,E1 -11244.907,E2 -11244.907} C_VEL
LIN {X 0,Y 395.779,Z 552.265,A -85,B 0,C 180,E1 -11245.927,E2 -11245.927} C_VEL
LIN {X 0,Y 395.764,Z 554.71,A -85,B 0,C 180,E1 -11247.965,E2 -11247.965} C_VEL
LIN {X 0,Y 395.792,Z 555.299,A -85,B 0,C 180,E1 -11248.983,E2 -11248.983} C_VEL
LIN {X 0,Y 395.792,Z 555.299,A -85,B 0,C 180,E1 -11251.017,E2 -11251.017} C_VEL
LIN {X 0,Y 395.764,Z 554.71,A -85,B 0,C 180,E1 -11252.035,E2 -11252.035} C_VEL
LIN {X 0,Y 395.779,Z 552.265,A -85,B 0,C 180,E1 -11254.073,E2 -11254.073} C_VEL
LIN {X 0,Y 395.851,Z 550.468,A -85,B 0,C 180,E1 -11255.093,E2 -11255.093} C_VEL
LIN {X 0,Y 395.921,Z 546.861,A -85,B 0,C 180,E1 -11256.625,E2 -11256.625} C_VEL
LIN {X 0,Y 396.228,Z 542.116,A -85,B 0,C 180,E1 -11258.157,E2 -11258.157} C_VEL
LIN {X 0,Y 396.629,Z 536.094,A -85,B 0,C 180,E1 -11259.691,E2 -11259.691} C_VEL
LIN {X 0,Y 397.073,Z 529.995,A -85,B 0,C 180,E1 -11260.968,E2 -11260.968} C_VEL
LIN {X 0,Y 397.604,Z 524.296,A -85,B 0,C 180,E1 -11261.987,E2 -11261.987} C_VEL
LIN {X 0,Y 398.329,Z 515.741,A -85,B 0,C 180,E1 -11263.26,E2 -11263.26} C_VEL
LIN {X 0,Y 398.954,Z 507.558,A -85,B 0,C 180,E1 -11264.278,E2 -11264.278} C_VEL
LIN {X 0,Y 399.621,Z 499.181,A -85,B 0,C 180,E1 -11265.152,E2 -11265.152} C_VEL
LIN {X 0,Y 400.33,Z 490.329,A -85,B 0,C 180,E1 -11265.92,E2 -11265.92} C_VEL
LIN {X 0,Y 400.921,Z 480.938,A -85,B 0,C 180,E1 -11266.591,E2 -11266.591} C_VEL
LIN {X 0,Y 399.779,Z 470.673,A -85,B 0,C 180,E1 -11267.244,E2 -11267.244} C_VEL
LIN {X 0,Y 397.973,Z 460.395,A -85,B 0,C 180,E1 -11267.786,E2 -11267.786} C_VEL
LIN {X 0,Y 395.953,Z 450.197,A -85,B 0,C 180,E1 -11268.226,E2 -11268.226} C_VEL
LIN {X 0,Y 396.102,Z 446.278,A -85,B 0,C 180,E1 -11270.784,E2 -11270.784} C_VEL
LIN {X 0,Y 396.335,Z 441.34,A -85,B 0,C 180,E1 -11274.069,E2 -11274.069} C_VEL
LIN {X 0,Y 396.685,Z 436.13,A -85,B 0,C 180,E1 -11277.644,E2 -11277.644} C_VEL
LIN {X 0,Y 397.021,Z 431.586,A -85,B 0,C 180,E1 -11280.887,E2 -11280.887} C_VEL
LIN {X 0,Y 397.407,Z 426.805,A -85,B 0,C 180,E1 -11284.464,E2 -11284.464} C_VEL
LIN {X 0,Y 397.756,Z 423.153,A -85,B 0,C 180,E1 -11287.334,E2 -11287.334} C_VEL
LIN {X 0,Y 398.064,Z 419.025,A -85,B 0,C 180,E1 -11290.786,E2 -11290.786} C_VEL
LIN {X 0,Y 398.076,Z 415.879,A -85,B 0,C 180,E1 -11293.626,E2 -11293.626} C_VEL
LIN {X 0,Y 397.749,Z 413.022,A -85,B 0,C 180,E1 -11296.44,E2 -11296.44} C_VEL
LIN {X 0,Y 397.358,Z 410.148,A -85,B 0,C 180,E1 -11299.51,E2 -11299.51} C_VEL
LIN {X 0,Y 397.142,Z 408.726,A -85,B 0,C 180,E1 -11301.135,E2 -11301.135} C_VEL
LIN {X 0,Y 397.116,Z 408.523,A -85,B 0,C 180,E1 -11304.496,E2 -11304.496} C_VEL
LIN {X 0,Y 397.107,Z 408.522,A -85,B 0,C 180,E1 -11307.93,E2 -11307.93} C_VEL
LIN {X 0,Y 397.122,Z 408.516,A -85,B 0,C 180,E1 -11311.456,E2 -11311.456} C_VEL
LIN {X 0,Y 397.147,Z 408.512,A -85,B 0,C 180,E1 -11314.487,E2 -11314.487} C_VEL
LIN {X 0,Y 397.089,Z 408.521,A -85,B 0,C 180,E1 -11318.181,E2 -11318.181} C_VEL
LIN {X 0,Y 397.156,Z 408.513,A -85,B 0,C 180,E1 -11321.426,E2 -11321.426} C_VEL
LIN {X 0,Y 397.177,Z 408.507,A -85,B 0,C 180,E1 -11324.607,E2 -11324.607} C_VEL
LIN {X 0,Y 397.212,Z 408.509,A -85,B 0,C 180,E1 -11327.741,E2 -11327.741} C_VEL
LIN {X 0,Y 397.245,Z 408.499,A -85,B 0,C 180,E1 -11330.837,E2 -11330.837} C_VEL
LIN {X 0,Y 397.366,Z 408.487,A -85,B 0,C 180,E1 -11333.908,E2 -11333.908} C_VEL
LIN {X 0,Y 397.444,Z 408.476,A -85,B 0,C 180,E1 -11337.973,E2 -11337.973} C_VEL
LIN {X 0,Y 397.572,Z 408.459,A -85,B 0,C 180,E1 -11339.999,E2 -11339.999} C_VEL
LIN {X 0,Y 397.374,Z 408.485,A -85,B 0,C 180,E1 -11343.041,E2 -11343.041} C_VEL
LIN {X 0,Y 397.339,Z 408.487,A -85,B 0,C 180,E1 -11346.644,E2 -11346.644} C_VEL
LIN {X 0,Y 397.244,Z 408.504,A -85,B 0,C 180,E1 -11349.161,E2 -11349.161} C_VEL
LIN {X 0,Y 397.211,Z 408.503,A -85,B 0,C 180,E1 -11352.258,E2 -11352.258} C_VEL
LIN {X 0,Y 397.171,Z 408.513,A -85,B 0,C 180,E1 -11355.392,E2 -11355.392} C_VEL
LIN {X 0,Y 397.153,Z 408.511,A -85,B 0,C 180,E1 -11358.573,E2 -11358.573} C_VEL
LIN {X 0,Y 397.088,Z 408.519,A -85,B 0,C 180,E1 -11361.818,E2 -11361.818} C_VEL
LIN {X 0,Y 397.148,Z 408.517,A -85,B 0,C 180,E1 -11365.132,E2 -11365.132} C_VEL
LIN {X 0,Y 397.155,Z 408.51,A -85,B 0,C 180,E1 -11367.776,E2 -11367.776} C_VEL
LIN {X 0,Y 397.077,Z 408.526,A -85,B 0,C 180,E1 -11370.882,E2 -11370.882} C_VEL
LIN {X 0,Y 397.117,Z 408.517,A -85,B 0,C 180,E1 -11374.493,E2 -11374.493} C_VEL
LIN {X 0,Y 397.102,Z 408.518,A -85,B 0,C 180,E1 -11378.274,E2 -11378.274} C_VEL
LIN {X 0,Y 397.148,Z 408.511,A -85,B 0,C 180,E1 -11381.993,E2 -11381.993} C_VEL
LIN {X 0,Y 397.106,Z 408.519,A -85,B 0,C 180,E1 -11385.065,E2 -11385.065} C_VEL
LIN {X 0,Y 397.061,Z 408.522,A -85,B 0,C 180,E1 -11388.021,E2 -11388.021} C_VEL
LIN {X 0,Y 397.127,Z 408.515,A -85,B 0,C 180,E1 -11391.138,E2 -11391.138} C_VEL
LIN {X 0,Y 397.114,Z 408.521,A -85,B 0,C 180,E1 -11394.497,E2 -11394.497} C_VEL
LIN {X 0,Y 397.072,Z 408.521,A -85,B 0,C 180,E1 -11397.929,E2 -11397.929} C_VEL
LIN {X 0,Y 397.116,Z 408.515,A -85,B 0,C 180,E1 -11401.457,E2 -11401.457} C_VEL
LIN {X 0,Y 397.148,Z 408.517,A -85,B 0,C 180,E1 -11404.488,E2 -11404.488} C_VEL
LIN {X 0,Y 397.104,Z 408.517,A -85,B 0,C 180,E1 -11407.086,E2 -11407.086} C_VEL
LIN {X 0,Y 397.143,Z 408.518,A -85,B 0,C 180,E1 -11410.353,E2 -11410.353} C_VEL
LIN {X 0,Y 397.162,Z 408.514,A -85,B 0,C 180,E1 -11413.553,E2 -11413.553} C_VEL
LIN {X 0,Y 397.224,Z 408.507,A -85,B 0,C 180,E1 -11416.703,E2 -11416.703} C_VEL
LIN {X 0,Y 397.214,Z 408.507,A -85,B 0,C 180,E1 -11419.809,E2 -11419.809} C_VEL
LIN {X 0,Y 397.361,Z 408.488,A -85,B 0,C 180,E1 -11422.888,E2 -11422.888} C_VEL
LIN {X 0,Y 397.252,Z 408.504,A -85,B 0,C 180,E1 -11424.925,E2 -11424.925} C_VEL
LIN {X 0,Y 397.448,Z 408.478,A -85,B 0,C 180,E1 -11427.973,E2 -11427.973} C_VEL
LIN {X 0,Y 397.577,Z 408.464,A -85,B 0,C 180,E1 -11430,E2 -11430} C_VEL
LIN {X 0,Y 397.378,Z 408.486,A -85,B 0,C 180,E1 -11433.041,E2 -11433.041} C_VEL
LIN {X 0,Y 397.361,Z 408.488,A -85,B 0,C 180,E1 -11437.112,E2 -11437.112} C_VEL
LIN {X 0,Y 397.214,Z 408.507,A -85,B 0,C 180,E1 -11440.191,E2 -11440.191} C_VEL
LIN {X 0,Y 397.222,Z 408.507,A -85,B 0,C 180,E1 -11443.321,E2 -11443.321} C_VEL
LIN {X 0,Y 397.177,Z 408.511,A -85,B 0,C 180,E1 -11447.155,E2 -11447.155} C_VEL
LIN {X 0,Y 397.104,Z 408.516,A -85,B 0,C 180,E1 -11450.729,E2 -11450.729} C_VEL
LIN {X 0,Y 397.128,Z 408.516,A -85,B 0,C 180,E1 -11454.018,E2 -11454.018} C_VEL
LIN {X 0,Y 397.129,Z 408.513,A -85,B 0,C 180,E1 -11456.329,E2 -11456.329} C_VEL
LIN {X 0,Y 396.459,Z 408.601,A -85,B 0,C 180,E1 -11457.176,E2 -11457.176} C_VEL
LIN {X 0,Y 393.584,Z 408.955,A -85,B 0,C 180,E1 -11458.551,E2 -11458.551} C_VEL
LIN {X 0,Y 391.145,Z 409.264,A -85,B 0,C 180,E1 -11459.663,E2 -11459.663} C_VEL
LIN {X 0,Y 390.094,Z 409.39,A -85,B 0,C 180,E1 -11460.522,E2 -11460.522} C_VEL
LIN {X 0,Y 390.006,Z 409.401,A -85,B 0,C 180,E1 -11460.814,E2 -11460.814} C_VEL
LIN {X 0,Y 390.062,Z 409.395,A -85,B 0,C 180,E1 -11464.024,E2 -11464.024} C_VEL
LIN {X 0,Y 390.039,Z 409.401,A -85,B 0,C 180,E1 -11467.551,E2 -11467.551} C_VEL
LIN {X 0,Y 390.05,Z 409.396,A -85,B 0,C 180,E1 -11470.821,E2 -11470.821} C_VEL
LIN {X 0,Y 390.05,Z 409.396,A -85,B 0,C 180,E1 -11473.886,E2 -11473.886} C_VEL
LIN {X 0,Y 390.052,Z 409.397,A -85,B 0,C 180,E1 -11476.79,E2 -11476.79} C_VEL
LIN {X 0,Y 390.048,Z 409.398,A -85,B 0,C 180,E1 -11479.56,E2 -11479.56} C_VEL
LIN {X 0,Y 390.037,Z 409.397,A -85,B 0,C 180,E1 -11482.449,E2 -11482.449} C_VEL
LIN {X 0,Y 390.06,Z 409.394,A -85,B 0,C 180,E1 -11486.045,E2 -11486.045} C_VEL
LIN {X 0,Y 390.044,Z 409.396,A -85,B 0,C 180,E1 -11489.868,E2 -11489.868} C_VEL
LIN {X 0,Y 390.105,Z 409.392,A -85,B 0,C 180,E1 -11493.232,E2 -11493.232} C_VEL
LIN {X 0,Y 390.098,Z 409.394,A -85,B 0,C 180,E1 -11496.751,E2 -11496.751} C_VEL
LIN {X 0,Y 390.095,Z 409.389,A -85,B 0,C 180,E1 -11499.983,E2 -11499.983} C_VEL
LIN {X 0,Y 390.129,Z 409.387,A -85,B 0,C 180,E1 -11503.248,E2 -11503.248} C_VEL
LIN {X 0,Y 390.186,Z 409.383,A -85,B 0,C 180,E1 -11506.562,E2 -11506.562} C_VEL
LIN {X 0,Y 390.196,Z 409.384,A -85,B 0,C 180,E1 -11510.672,E2 -11510.672} C_VEL
LIN {X 0,Y 390.32,Z 409.361,A -85,B 0,C 180,E1 -11513.799,E2 -11513.799} C_VEL
LIN {X 0,Y 390.412,Z 409.351,A -85,B 0,C 180,E1 -11517.937,E2 -11517.937} C_VEL
LIN {X 0,Y 390.542,Z 409.335,A -85,B 0,C 180,E1 -11520.001,E2 -11520.001} C_VEL
LIN {X 0,Y 390.308,Z 409.364,A -85,B 0,C 180,E1 -11523.097,E2 -11523.097} C_VEL
LIN {X 0,Y 390.32,Z 409.365,A -85,B 0,C 180,E1 -11526.203,E2 -11526.203} C_VEL
LIN {X 0,Y 390.198,Z 409.376,A -85,B 0,C 180,E1 -11529.33,E2 -11529.33} C_VEL
LIN {X 0,Y 390.188,Z 409.378,A -85,B 0,C 180,E1 -11533.439,E2 -11533.439} C_VEL
LIN {X 0,Y 390.144,Z 409.383,A -85,B 0,C 180,E1 -11537.309,E2 -11537.309} C_VEL
LIN {X 0,Y 390.081,Z 409.395,A -85,B 0,C 180,E1 -11540.471,E2 -11540.471} C_VEL
LIN {X 0,Y 390.067,Z 409.393,A -85,B 0,C 180,E1 -11543.353,E2 -11543.353} C_VEL
LIN {X 0,Y 390.108,Z 409.388,A -85,B 0,C 180,E1 -11546.769,E2 -11546.769} C_VEL
LIN {X 0,Y 390.04,Z 409.4,A -85,B 0,C 180,E1 -11550.3,E2 -11550.3} C_VEL
LIN {X 0,Y 390.081,Z 409.398,A -85,B 0,C 180,E1 -11553.954,E2 -11553.954} C_VEL
LIN {X 0,Y 390.044,Z 409.402,A -85,B 0,C 180,E1 -11557.552,E2 -11557.552} C_VEL
LIN {X 0,Y 390.194,Z 410.203,A -85,B 0,C 180,E1 -11559.242,E2 -11559.242} C_VEL
LIN {X 0,Y 390.602,Z 413.079,A -85,B 0,C 180,E1 -11562.465,E2 -11562.465} C_VEL
LIN {X 0,Y 391.012,Z 416.52,A -85,B 0,C 180,E1 -11565.969,E2 -11565.969} C_VEL
LIN {X 0,Y 391.031,Z 419.804,A -85,B 0,C 180,E1 -11569.014,E2 -11569.014} C_VEL
LIN {X 0,Y 390.748,Z 423.658,A -85,B 0,C 180,E1 -11572.316,E2 -11572.316} C_VEL
LIN {X 0,Y 390.314,Z 428.335,A -85,B 0,C 180,E1 -11576.07,E2 -11576.07} C_VEL
LIN {X 0,Y 390.024,Z 431.514,A -85,B 0,C 180,E1 -11578.497,E2 -11578.497} C_VEL
LIN {X 0,Y 389.631,Z 436.45,A -85,B 0,C 180,E1 -11582.11,E2 -11582.11} C_VEL
LIN {X 0,Y 389.28,Z 441.223,A -85,B 0,C 180,E1 -11585.466,E2 -11585.466} C_VEL
LIN {X 0,Y 389.046,Z 446.155,A -85,B 0,C 180,E1 -11588.821,E2 -11588.821} C_VEL
LIN {X 0,Y 388.888,Z 450.007,A -85,B 0,C 180,E1 -11591.427,E2 -11591.427} C_VEL
LIN {X 0,Y 392.052,Z 466.343,A -85,B 0,C 180,E1 -11592.19,E2 -11592.19} C_VEL
LIN {X 0,Y 393.555,Z 476.582,A -85,B 0,C 180,E1 -11592.814,E2 -11592.814} C_VEL
LIN {X 0,Y 394.08,Z 482.476,A -85,B 0,C 180,E1 -11593.227,E2 -11593.227} C_VEL
LIN {X 0,Y 393.166,Z 494.794,A -85,B 0,C 180,E1 -11594.181,E2 -11594.181} C_VEL
LIN {X 0,Y 392.295,Z 505.096,A -85,B 0,C 180,E1 -11595.21,E2 -11595.21} C_VEL
LIN {X 0,Y 391.52,Z 513.855,A -85,B 0,C 180,E1 -11596.273,E2 -11596.273} C_VEL
LIN {X 0,Y 390.943,Z 520.844,A -85,B 0,C 180,E1 -11597.278,E2 -11597.278} C_VEL
LIN {X 0,Y 390.324,Z 527.045,A -85,B 0,C 180,E1 -11598.313,E2 -11598.313} C_VEL
LIN {X 0,Y 389.803,Z 533.585,A -85,B 0,C 180,E1 -11599.613,E2 -11599.613} C_VEL
LIN {X 0,Y 389.445,Z 538.087,A -85,B 0,C 180,E1 -11600.653,E2 -11600.653} C_VEL
LIN {X 0,Y 389.044,Z 543.578,A -85,B 0,C 180,E1 -11602.213,E2 -11602.213} C_VEL
LIN {X 0,Y 388.796,Z 547.902,A -85,B 0,C 180,E1 -11603.774,E2 -11603.774} C_VEL
LIN {X 0,Y 388.747,Z 550.27,A -85,B 0,C 180,E1 -11604.814,E2 -11604.814} C_VEL
LIN {X 0,Y 388.704,Z 552.068,A -85,B 0,C 180,E1 -11605.853,E2 -11605.853} C_VEL
LIN {X 0,Y 388.662,Z 554.513,A -85,B 0,C 180,E1 -11607.927,E2 -11607.927} C_VEL
LIN {X 0,Y 388.704,Z 555.102,A -85,B 0,C 180,E1 -11608.964,E2 -11608.964} C_VEL
LIN {X 0,Y 388.704,Z 555.102,A -85,B 0,C 180,E1 -11611.036,E2 -11611.036} C_VEL
LIN {X 0,Y 388.662,Z 554.513,A -85,B 0,C 180,E1 -11612.073,E2 -11612.073} C_VEL
LIN {X 0,Y 388.704,Z 552.068,A -85,B 0,C 180,E1 -11614.147,E2 -11614.147} C_VEL
LIN {X 0,Y 388.732,Z 548.995,A -85,B 0,C 180,E1 -11615.759,E2 -11615.759} C_VEL
LIN {X 0,Y 388.942,Z 545.132,A -85,B 0,C 180,E1 -11617.266,E2 -11617.266} C_VEL
LIN {X 0,Y 389.299,Z 540.003,A -85,B 0,C 180,E1 -11618.827,E2 -11618.827} C_VEL
LIN {X 0,Y 389.676,Z 534.74,A -85,B 0,C 180,E1 -11620.128,E2 -11620.128} C_VEL
LIN {X 0,Y 390.183,Z 528.421,A -85,B 0,C 180,E1 -11621.428,E2 -11621.428} C_VEL
LIN {X 0,Y 390.774,Z 522.471,A -85,B 0,C 180,E1 -11622.463,E2 -11622.463} C_VEL
LIN {X 0,Y 391.385,Z 515.543,A -85,B 0,C 180,E1 -11623.499,E2 -11623.499} C_VEL
LIN {X 0,Y 392.026,Z 507.36,A -85,B 0,C 180,E1 -11624.535,E2 -11624.535} C_VEL
LIN {X 0,Y 392.752,Z 498.848,A -85,B 0,C 180,E1 -11625.437,E2 -11625.437} C_VEL
LIN {X 0,Y 393.504,Z 490.132,A -85,B 0,C 180,E1 -11626.204,E2 -11626.204} C_VEL
LIN {X 0,Y 394.055,Z 482.48,A -85,B 0,C 180,E1 -11626.774,E2 -11626.774} C_VEL
LIN {X 0,Y 392.971,Z 471.884,A -85,B 0,C 180,E1 -11627.479,E2 -11627.479} C_VEL
LIN {X 0,Y 391.141,Z 461.251,A -85,B 0,C 180,E1 -11628.066,E2 -11628.066} C_VEL
LIN {X 0,Y 388.885,Z 450.012,A -85,B 0,C 180,E1 -11628.57,E2 -11628.57} C_VEL
LIN {X 0,Y 389.046,Z 446.136,A -85,B 0,C 180,E1 -11631.179,E2 -11631.179} C_VEL
LIN {X 0,Y 389.279,Z 441.21,A -85,B 0,C 180,E1 -11634.534,E2 -11634.534} C_VEL
LIN {X 0,Y 389.637,Z 436.333,A -85,B 0,C 180,E1 -11637.967,E2 -11637.967} C_VEL
LIN {X 0,Y 390.026,Z 431.506,A -85,B 0,C 180,E1 -11641.503,E2 -11641.503} C_VEL
LIN {X 0,Y 390.448,Z 426.756,A -85,B 0,C 180,E1 -11645.168,E2 -11645.168} C_VEL
LIN {X 0,Y 390.749,Z 423.622,A -85,B 0,C 180,E1 -11647.699,E2 -11647.699} C_VEL
LIN {X 0,Y 391.031,Z 419.797,A -85,B 0,C 180,E1 -11650.986,E2 -11650.986} C_VEL
LIN {X 0,Y 391.063,Z 417.506,A -85,B 0,C 180,E1 -11653.071,E2 -11653.071} C_VEL
LIN {X 0,Y 390.788,Z 414.54,A -85,B 0,C 180,E1 -11656.001,E2 -11656.001} C_VEL
LIN {X 0,Y 390.355,Z 411.207,A -85,B 0,C 180,E1 -11659.597,E2 -11659.597} C_VEL
LIN {X 0,Y 390.162,Z 410.068,A -85,B 0,C 180,E1 -11660.916,E2 -11660.916} C_VEL
LIN {X 0,Y 390.044,Z 409.403,A -85,B 0,C 180,E1 -11662.448,E2 -11662.448} C_VEL
LIN {X 0,Y 390.081,Z 409.398,A -85,B 0,C 180,E1 -11666.046,E2 -11666.046} C_VEL
LIN {X 0,Y 390.04,Z 409.4,A -85,B 0,C 180,E1 -11669.7,E2 -11669.7} C_VEL
LIN {X 0,Y 390.108,Z 409.388,A -85,B 0,C 180,E1 -11673.231,E2 -11673.231} C_VEL
LIN {X 0,Y 390.071,Z 409.392,A -85,B 0,C 180,E1 -11676.76,E2 -11676.76} C_VEL
LIN {X 0,Y 390.098,Z 409.394,A -85,B 0,C 180,E1 -11679.982,E2 -11679.982} C_VEL
LIN {X 0,Y 390.135,Z 409.386,A -85,B 0,C 180,E1 -11683.248,E2 -11683.248} C_VEL
LIN {X 0,Y 390.188,Z 409.378,A -85,B 0,C 180,E1 -11686.561,E2 -11686.561} C_VEL
LIN {X 0,Y 390.198,Z 409.376,A -85,B 0,C 180,E1 -11690.67,E2 -11690.67} C_VEL
LIN {X 0,Y 390.32,Z 409.365,A -85,B 0,C 180,E1 -11693.797,E2 -11693.797} C_VEL
LIN {X 0,Y 390.412,Z 409.352,A -85,B 0,C 180,E1 -11697.936,E2 -11697.936} C_VEL
LIN {X 0,Y 390.542,Z 409.335,A -85,B 0,C 180,E1 -11699.999,E2 -11699.999} C_VEL
LIN {X 0,Y 390.308,Z 409.366,A -85,B 0,C 180,E1 -11703.096,E2 -11703.096} C_VEL
LIN {X 0,Y 390.294,Z 409.365,A -85,B 0,C 180,E1 -11706.639,E2 -11706.639} C_VEL
LIN {X 0,Y 390.196,Z 409.384,A -85,B 0,C 180,E1 -11709.328,E2 -11709.328} C_VEL
LIN {X 0,Y 390.186,Z 409.383,A -85,B 0,C 180,E1 -11713.438,E2 -11713.438} C_VEL
LIN {X 0,Y 390.14,Z 409.389,A -85,B 0,C 180,E1 -11717.307,E2 -11717.307} C_VEL
LIN {X 0,Y 390.078,Z 409.392,A -85,B 0,C 180,E1 -11720.47,E2 -11720.47} C_VEL
LIN {X 0,Y 390.081,Z 409.395,A -85,B 0,C 180,E1 -11723.351,E2 -11723.351} C_VEL
LIN {X 0,Y 390.105,Z 409.392,A -85,B 0,C 180,E1 -11726.768,E2 -11726.768} C_VEL
LIN {X 0,Y 390.036,Z 409.397,A -85,B 0,C 180,E1 -11730.299,E2 -11730.299} C_VEL
LIN {X 0,Y 390.06,Z 409.394,A -85,B 0,C 180,E1 -11734.025,E2 -11734.025} C_VEL
LIN {X 0,Y 390.039,Z 409.397,A -85,B 0,C 180,E1 -11737.552,E2 -11737.552} C_VEL
LIN {X 0,Y 390.075,Z 409.398,A -85,B 0,C 180,E1 -11740.826,E2 -11740.826} C_VEL
LIN {X 0,Y 390.095,Z 409.389,A -85,B 0,C 180,E1 -11743.894,E2 -11743.894} C_VEL
LIN {X 0,Y 390.037,Z 409.396,A -85,B 0,C 180,E1 -11747.626,E2 -11747.626} C_VEL
LIN {X 0,Y 390.086,Z 409.394,A -85,B 0,C 180,E1 -11750.908,E2 -11750.908} C_VEL
LIN {X 0,Y 390.079,Z 409.396,A -85,B 0,C 180,E1 -11754.793,E2 -11754.793} C_VEL
LIN {X 0,Y 390.018,Z 409.406,A -85,B 0,C 180,E1 -11758.496,E2 -11758.496} C_VEL
LIN {X 0,Y 390.112,Z 409.39,A -85,B 0,C 180,E1 -11762.07,E2 -11762.07} C_VEL
LIN {X 0,Y 390.075,Z 409.392,A -85,B 0,C 180,E1 -11765.52,E2 -11765.52} C_VEL
LIN {X 0,Y 390.051,Z 409.399,A -85,B 0,C 180,E1 -11768.878,E2 -11768.878} C_VEL
LIN {X 0,Y 390.123,Z 409.392,A -85,B 0,C 180,E1 -11772.167,E2 -11772.167} C_VEL
LIN {X 0,Y 390.14,Z 409.388,A -85,B 0,C 180,E1 -11775.393,E2 -11775.393} C_VEL
LIN {X 0,Y 390.145,Z 409.389,A -85,B 0,C 180,E1 -11778.571,E2 -11778.571} C_VEL
LIN {X 0,Y 390.318,Z 409.368,A -85,B 0,C 180,E1 -11782.535,E2 -11782.535} C_VEL
LIN {X 0,Y 390.35,Z 409.568,A -85,B 0,C 180,E1 -11782.704,E2 -11782.704} C_VEL
LIN {X 0,Y 390.912,Z 411.477,A -85,B 0,C 180,E1 -11783.16,E2 -11783.16} C_VEL
LIN {X 0,Y 392.539,Z 413.758,A -85,B 0,C 180,E1 -11784.349,E2 -11784.349} C_VEL
LIN {X 0,Y 394.308,Z 415.018,A -85,B 0,C 180,E1 -11785.912,E2 -11785.912} C_VEL
LIN {X 0,Y 395.197,Z 415.227,A -85,B 0,C 180,E1 -11786.942,E2 -11786.942} C_VEL
LIN {X 0,Y 396.207,Z 415.465,A -85,B 0,C 180,E1 -11788.984,E2 -11788.984} C_VEL
LIN {X 0,Y 396.373,Z 415.461,A -85,B 0,C 180,E1 -11790,E2 -11790} C_VEL
LIN {X 0,Y 395.808,Z 415.385,A -85,B 0,C 180,E1 -11792.035,E2 -11792.035} C_VEL
LIN {X 0,Y 394.474,Z 415.067,A -85,B 0,C 180,E1 -11793.894,E2 -11793.894} C_VEL
LIN {X 0,Y 392.691,Z 413.906,A -85,B 0,C 180,E1 -11795.52,E2 -11795.52} C_VEL
LIN {X 0,Y 390.995,Z 411.652,A -85,B 0,C 180,E1 -11796.774,E2 -11796.774} C_VEL
LIN {X 0,Y 390.384,Z 409.733,A -85,B 0,C 180,E1 -11797.267,E2 -11797.267} C_VEL
LIN {X 0,Y 390.316,Z 409.367,A -85,B 0,C 180,E1 -11797.353,E2 -11797.353} C_VEL
LIN {X 0,Y 390.165,Z 409.385,A -85,B 0,C 180,E1 -11800.377,E2 -11800.377} C_VEL
LIN {X 0,Y 390.165,Z 409.387,A -85,B 0,C 180,E1 -11803.542,E2 -11803.542} C_VEL
LIN {X 0,Y 390.144,Z 409.388,A -85,B 0,C 180,E1 -11807.308,E2 -11807.308} C_VEL
LIN {X 0,Y 390.083,Z 409.391,A -85,B 0,C 180,E1 -11810.47,E2 -11810.47} C_VEL
LIN {X 0,Y 390.084,Z 409.394,A -85,B 0,C 180,E1 -11813.351,E2 -11813.351} C_VEL
LIN {X 0,Y 390.108,Z 409.388,A -85,B 0,C 180,E1 -11816.768,E2 -11816.768} C_VEL
LIN {X 0,Y 390.033,Z 409.397,A -85,B 0,C 180,E1 -11820.299,E2 -11820.299} C_VEL
LIN {X 0,Y 390.006,Z 409.401,A -85,B 0,C 180,E1 -11820.814,E2 -11820.814} C_VEL
LIN {X 0,Y 389.333,Z 409.489,A -85,B 0,C 180,E1 -11821.676,E2 -11821.676} C_VEL
LIN {X 0,Y 386.485,Z 409.842,A -85,B 0,C 180,E1 -11823.078,E2 -11823.078} C_VEL
LIN {X 0,Y 384.087,Z 410.138,A -85,B 0,C 180,E1 -11824.21,E2 -11824.21} C_VEL
LIN {X 0,Y 383.069,Z 410.267,A -85,B 0,C 180,E1 -11825.086,E2 -11825.086} C_VEL
LIN {X 0,Y 382.992,Z 410.272,A -85,B 0,C 180,E1 -11825.383,E2 -11825.383} C_VEL
LIN {X 0,Y 382.999,Z 410.274,A -85,B 0,C 180,E1 -11828.6,E2 -11828.6} C_VEL
LIN {X 0,Y 382.979,Z 410.282,A -85,B 0,C 180,E1 -11831.347,E2 -11831.347} C_VEL
LIN {X 0,Y 382.992,Z 410.274,A -85,B 0,C 180,E1 -11834.304,E2 -11834.304} C_VEL
LIN {X 0,Y 383.002,Z 410.28,A -85,B 0,C 180,E1 -11837.24,E2 -11837.24} C_VEL
LIN {X 0,Y 383.007,Z 410.273,A -85,B 0,C 180,E1 -11840.413,E2 -11840.413} C_VEL
